(* IEC 61131-3 sources: SmartHomeNew/snapshots/2026-05-04 (part 2) *)

(* ---- FB_System_Timebase.st ---- *)
// ==============================================================================
// System timebase helper
//
// Internal helper for PRG_System.
// Owns PLC runtime clock projection into GVL_STATUS:
// - monotonic system milliseconds
// - time-of-day milliseconds
// - day of week / day of year rollover
// - TOD representation
// ==============================================================================
FUNCTION_BLOCK FB_System_Timebase
VAR
    L_Time_Diff : UDINT;
END_VAR

GVL_STATUS.G_System_Time_MS := TIME_TO_UDINT(TIME());

L_Time_Diff := SEL(
    GVL_STATUS.G_System_Time_MS >= GVL_STATUS.G_Last_System_Time_MS,
    GVL_STATUS.G_System_Time_MS - GVL_STATUS.G_Last_System_Time_MS,
    (4294967295 - GVL_STATUS.G_Last_System_Time_MS) + GVL_STATUS.G_System_Time_MS + 1
);

GVL_STATUS.G_Time_Of_Day_MS := (GVL_STATUS.G_Time_Of_Day_MS + L_Time_Diff) MOD 86400000;

IF GVL_STATUS.G_Time_Of_Day_MS < L_Time_Diff THEN
    GVL_STATUS.G_Current_Day := (GVL_STATUS.G_Current_Day MOD 7) + 1;
    GVL_STATUS.G_Day_Of_Year := (GVL_STATUS.G_Day_Of_Year MOD 365) + 1;
END_IF;

GVL_STATUS.G_Last_System_Time_MS := GVL_STATUS.G_System_Time_MS;
GVL_STATUS.G_Current_TOD := UDINT_TO_TOD(GVL_STATUS.G_Time_Of_Day_MS);

// >>> BULK_SYNC_ANCHOR: FB_System_Timebase <<<

(* ---- FB_Test_Result_Handler.st ---- *)
FUNCTION_BLOCK FB_Test_Result_Handler
VAR_INPUT
    VI_Test_Passed : BOOL;
END_VAR
VAR
    L_Latched_Failure : BOOL;
END_VAR

// latch failure
IF NOT VI_Test_Passed THEN
    L_Latched_Failure := TRUE;
END_IF;

// enforce safe stop if failure latched
IF L_Latched_Failure THEN
    GVL_COMMAND.G_Gas_Valve_Close := TRUE;
    GVL_COMMAND.G_Close_Valve_35 := TRUE;
    GVL_COMMAND.G_Close_Valve_36 := TRUE;
END_IF;
END_FUNCTION_BLOCK

(* ---- FB_Trend_Adapter.st ---- *)
FUNCTION_BLOCK FB_Trend_Adapter
VAR_INPUT
    VI_Data : ST_Trend_Data;
END_VAR

VAR_OUTPUT
    VO_Average : REAL;
    VO_Min : REAL;
    VO_Max : REAL;
    VO_Trend_Up : BOOL;
    VO_Trend_Down : BOOL;
END_VAR

VAR
    fbAnalyzer : FB_Trend_Analyzer;
    L_Data_Copy : ARRAY[1..GVL_CONSTANTS.C_MAX_TREND_DATA_POINTS] OF REAL;
    L_Count : INT;
    L_i : INT;
END_VAR

// Normalize count to analyzer bounds
L_Count := UDINT_TO_INT(VI_Data.record_count);
IF L_Count < 0 THEN
    L_Count := 0;
END_IF;
IF L_Count > GVL_CONSTANTS.C_MAX_TREND_DATA_POINTS THEN
    L_Count := GVL_CONSTANTS.C_MAX_TREND_DATA_POINTS;
END_IF;

// Copy source values into analyzer-compatible buffer
FOR L_i := 1 TO GVL_CONSTANTS.C_MAX_TREND_DATA_POINTS DO
    L_Data_Copy[L_i] := 0.0;
END_FOR;

IF L_Count > 0 THEN
    FOR L_i := 1 TO L_Count DO
        L_Data_Copy[L_i] := VI_Data.values[L_i];
    END_FOR;
END_IF;

fbAnalyzer(
    VI_Count := L_Count,
    VI_Data := L_Data_Copy,
    VO_Average => VO_Average,
    VO_Max => VO_Max,
    VO_Min => VO_Min,
    VO_Trend_Up => VO_Trend_Up,
    VO_Trend_Down => VO_Trend_Down
);
END_FUNCTION_BLOCK

(* ---- FB_Trend_Analyzer.st ---- *)
FUNCTION_BLOCK FB_Trend_Analyzer
VAR_INPUT
    VI_Count      : INT;
END_VAR
VAR_IN_OUT
    VI_Data       : ARRAY[1..GVL_CONSTANTS.C_MAX_TREND_DATA_POINTS] OF REAL;
END_VAR
VAR_OUTPUT
    VO_Average    : REAL;
    VO_Max        : REAL;
    VO_Min        : REAL;
    VO_Trend_Up   : BOOL;
    VO_Trend_Down : BOOL;
END_VAR
VAR
    L_i   : INT;
    L_Sum : REAL;
END_VAR

IF VI_Count > 0 AND VI_Count <= GVL_CONSTANTS.C_MAX_TREND_DATA_POINTS THEN
    VO_Max := VI_Data[1];
    VO_Min := VI_Data[1];
    L_Sum := 0.0;

    FOR L_i := 1 TO VI_Count DO
        IF VI_Data[L_i] > VO_Max THEN VO_Max := VI_Data[L_i]; END_IF;
        IF VI_Data[L_i] < VO_Min THEN VO_Min := VI_Data[L_i]; END_IF;
        L_Sum := L_Sum + VI_Data[L_i];
    END_FOR;

    VO_Average := L_Sum / INT_TO_REAL(VI_Count);

    IF VI_Count >= 2 THEN
        VO_Trend_Up := (VI_Data[VI_Count] > VI_Data[1]);
        VO_Trend_Down := (VI_Data[VI_Count] < VI_Data[1]);
    END_IF;
END_IF;
END_FUNCTION_BLOCK

(* ---- FB_Ventilation_System_Manager.st ---- *)
FUNCTION_BLOCK FB_Ventilation_System_Manager
VAR_INPUT
    VI_System_Time_MS : UDINT; // Системное время (мс)
    VI_IsActivePLC : BOOL; // Флаг: Данный ПЛК является ведущим
    VI_Outdoor_Temp : REAL; // Уличная температура воздуха (°C)
    VI_Current_Scenario : E_SCENARIO_TYPE; // Текущий глобальный сценарий
    VI_System_Mode : E_System_Operating_Mode; // Агрегированный режим работы системы
    VI_Config : ST_Ventilation_Global_Config; // Конфигурация системы вентиляции
    VI_Fire_Alarm : BOOL; // Сигнал пожарной тревоги
    VI_Gas_Alarm : BOOL; // Сигнал газовой тревоги
    VI_PV3_Boost_Req : BOOL; // Запрос форсирования ПВ-3 от газоанализатора (ТЗ 5.1)
    VI_Supply_100_Req : BOOL; // Запрос 100% притока (ТЗ 6.4)
    VI_Exhaust_100_Req : BOOL; // Запрос 100% вытяжки (ТЗ 6.4)
    VI_Supply_80_Req : BOOL; // Запрос 80% притока (ТЗ 5.4)
    VI_Vent_Stop : BOOL; // Запрос на остановку вентиляции (ТЗ 5.3)
    VI_IO_Modules_Online : ARRAY[1..GVL_CONSTANTS.C_MAX_MODULES] OF BOOL; // Статусы модулей ввода-вывода (только чтение)
END_VAR
VAR_IN_OUT
    VI_Supply_Temps : ARRAY[1..GVL_CONSTANTS.C_MAX_SUPPLY_TEMPS] OF REAL; // Температура приточного воздуха после калорифера
    VI_Room_Temps : ARRAY[1..16] OF REAL; // Температура в помещениях (°C)
    VI_Room_Humidities : ARRAY[1..16] OF REAL; // Влажность в помещениях (%)
    VI_Room_CO2 : ARRAY[1..16] OF REAL; // Уровень CO2 в помещениях (ppm)
    VI_Wet_Zone_Active : ARRAY[1..GVL_CONSTANTS.C_MAX_WET_ZONES] OF BOOL; // Сигналы включения света в санузлах (ТЗ 4.0)
    VI_Rule_Actions : ARRAY[1..GVL_CONSTANTS.C_MAX_RULES] OF ST_Rule_Action; // Действия от Rule Engine
END_VAR
VAR_OUTPUT
    VO_Supply_Fans : ARRAY[1..GVL_CONSTANTS.C_MAX_SUPPLY_FANS] OF BYTE; // Выход: Управление приточными вентиляторами (0-100%)
    VO_Exhaust_Fans : ARRAY[1..GVL_CONSTANTS.C_MAX_EXHAUST_FANS] OF BYTE; // Выход: Управление вытяжными вентиляторами (0-100%)
    VO_Heater_Power : ARRAY[1..GVL_CONSTANTS.C_MAX_BOILERS] OF REAL; // Выход: Мощность калориферов (0-100%)
    VO_Status_Msg : STRING(200); // Строковое сообщение о статусе
    VO_Ventilation_IO_Fault : BOOL; // Выход: диагностика потери связи с модулями ввода-вывода
    VO_Ventilation_Subsystem_Degraded : BOOL; // Выход: признак degraded-состояния подсистемы вентиляции
END_VAR
VAR
    L_Policy_Normal : BOOL;
    L_Policy_Safe_Stop : BOOL;
    L_Policy_Degraded : BOOL;
    L_Policy_Freeze_Protection : BOOL;
    L_i : INT;
    L_j : INT;
    L_Max_CO2 : REAL;
    L_Max_Hum : REAL;
    L_Base_Speed : BYTE;
    L_Target_Temp : REAL;
    L_PID_Heaters : ARRAY[1..GVL_CONSTANTS.C_MAX_BOILERS] OF FB_PID_Controller;
    L_Wet_Zone_Timers : ARRAY[1..GVL_CONSTANTS.C_MAX_WET_ZONES] OF FB_System_Timer_TOF; // Таймеры выбега для вытяжек санузлов
END_VAR

// ========================================
// Ventilation policy layer
// ========================================
VO_Ventilation_IO_Fault := FALSE;
VO_Ventilation_Subsystem_Degraded := FALSE;
L_Policy_Normal := (VI_System_Mode = E_System_Operating_Mode.MODE_NORMAL);
L_Policy_Safe_Stop := (VI_System_Mode = E_System_Operating_Mode.MODE_SAFE_STOP);
L_Policy_Degraded := (VI_System_Mode = E_System_Operating_Mode.MODE_DEGRADED);
L_Policy_Freeze_Protection := (VI_System_Mode = E_System_Operating_Mode.MODE_FREEZE_PROTECTION);

IF NOT VI_IsActivePLC THEN
    FOR L_i := 1 TO GVL_CONSTANTS.C_MAX_SUPPLY_FANS DO
        VO_Supply_Fans[L_i] := 0;
        IF L_i <= GVL_CONSTANTS.C_MAX_SUPPLY_TEMPS THEN
            VO_Heater_Power[L_i] := 0.0;
        END_IF;
    END_FOR;
    FOR L_i := 1 TO GVL_CONSTANTS.C_MAX_EXHAUST_FANS DO
        VO_Exhaust_Fans[L_i] := 0;
    END_FOR;
    VO_Status_Msg := 'ВЕНТИЛЯЦИЯ: РЕЗЕРВНЫЙ ПЛК';
    RETURN;
END_IF;

// Проверка связи с модулями ввода-вывода
FOR L_i := 1 TO GVL_CONSTANTS.C_MAX_MODULES DO
    IF NOT VI_IO_Modules_Online[L_i] THEN
        VO_Ventilation_IO_Fault := TRUE;
        // Переход в безопасное состояние при потере связи (отключение вентиляции)
        FOR L_j := 1 TO GVL_CONSTANTS.C_MAX_SUPPLY_FANS DO
            VO_Supply_Fans[L_j] := 0;
        END_FOR;
        FOR L_j := 1 TO GVL_CONSTANTS.C_MAX_EXHAUST_FANS DO
            VO_Exhaust_Fans[L_j] := 0;
        END_FOR;
        FOR L_j := 1 TO GVL_CONSTANTS.C_MAX_BOILERS DO
            VO_Heater_Power[L_j] := 0.0;
        END_FOR;
        VO_Status_Msg := 'ОШИБКА: Потеря связи с модулями ввода-вывода';
        RETURN;
    END_IF;
END_FOR;

// =========================
// SYSTEM MODE OVERRIDE
// =========================
// VENT_POLICY_ROUTING_PHASE3_V2
IF L_Policy_Safe_Stop THEN
    FOR L_i := 1 TO GVL_CONSTANTS.C_MAX_SUPPLY_FANS DO
        VO_Supply_Fans[L_i] := 0;
    END_FOR;
    FOR L_i := 1 TO GVL_CONSTANTS.C_MAX_EXHAUST_FANS DO
        VO_Exhaust_Fans[L_i] := 0;
    END_FOR;
    FOR L_i := 1 TO GVL_CONSTANTS.C_MAX_BOILERS DO
        VO_Heater_Power[L_i] := 0.0;
    END_FOR;
    VO_Status_Msg := 'ВЕНТИЛЯЦИЯ: ОСТАНОВЛЕНА POLICY SAFE_STOP';
    RETURN;
END_IF;

IF L_Policy_Degraded THEN
    FOR L_i := 1 TO GVL_CONSTANTS.C_MAX_SUPPLY_FANS DO
        VO_Supply_Fans[L_i] := 0;
    END_FOR;
    FOR L_i := 1 TO GVL_CONSTANTS.C_MAX_BOILERS DO
        VO_Heater_Power[L_i] := 0.0;
    END_FOR;
    VO_Ventilation_Subsystem_Degraded := TRUE;
    VO_Status_Msg := 'ВЕНТИЛЯЦИЯ: DEGRADED POLICY';
END_IF;

IF L_Policy_Freeze_Protection THEN
    FOR L_i := 1 TO GVL_CONSTANTS.C_MAX_SUPPLY_FANS DO
        VO_Supply_Fans[L_i] := 0;
    END_FOR;
    FOR L_i := 1 TO GVL_CONSTANTS.C_MAX_EXHAUST_FANS DO
        VO_Exhaust_Fans[L_i] := 0;
    END_FOR;
    FOR L_i := 1 TO GVL_CONSTANTS.C_MAX_BOILERS DO
        VO_Heater_Power[L_i] := 0.0;
    END_FOR;
    VO_Status_Msg := 'ВЕНТИЛЯЦИЯ: FREEZE_PROTECTION POLICY (stop)';
    RETURN;
END_IF;

// MODE_FREEZE_PROTECTION пока оставляем на текущей штатной логике

// 1. Определение базовой скорости и целевой температуры по сценарию (ТЗ 7.1)
CASE VI_Current_Scenario OF
    E_SCENARIO_TYPE.SCENARIO_AWAY:
        L_Base_Speed := VI_Config.Scenario_Modes[3].Base_Fan_Speed;
        L_Target_Temp := VI_Config.Scenario_Modes[3].Target_Temp;
    E_SCENARIO_TYPE.SCENARIO_SLEEP:
        L_Base_Speed := VI_Config.Scenario_Modes[2].Base_Fan_Speed;
        L_Target_Temp := VI_Config.Scenario_Modes[2].Target_Temp;
    ELSE // PRESENCE, MORNING, EVENING
        L_Base_Speed := VI_Config.Scenario_Modes[1].Base_Fan_Speed;
        L_Target_Temp := VI_Config.Scenario_Modes[1].Target_Temp;
END_CASE;

// 2. Логика управления приточными установками (П-1, П-2, П-3)
FOR L_i := 1 TO GVL_CONSTANTS.C_MAX_SUPPLY_FANS DO
    // ПИД-регулирование мощности электрического калорифера
    IF L_i <= GVL_CONSTANTS.C_MAX_SUPPLY_TEMPS THEN
        L_PID_Heaters[L_i](
            VI_SetPoint := L_Target_Temp,
            VI_ProcessValue := VI_Supply_Temps[L_i], // Используем датчик температуры после калорифера
            VI_Kp := 4.0, VI_Tn := 120.0, VI_Tv := 0.0,
            VI_Y_Min := 0.0, VI_Y_Max := 100.0, VI_Cycle_Time_S := 1.0,
            VO_Output => VO_Heater_Power[L_i]
        );
    END_IF;

    // Определение скорости приточного вентилятора
    VO_Supply_Fans[L_i] := L_Base_Speed;

    // Обработка действий от Rule Engine
    FOR L_j := 1 TO GVL_CONSTANTS.C_MAX_RULES DO
        IF VI_Rule_Actions[L_j].Active AND VI_Rule_Actions[L_j].Target_ID = L_i THEN
            IF VI_Rule_Actions[L_j].Action_Type = E_Rule_Action_Type.ACTION_SET_VENTILATION THEN
                VO_Supply_Fans[L_i] := REAL_TO_BYTE(VI_Rule_Actions[L_j].Value);
            END_IF;
        END_IF;
    END_FOR;

    // Requests are operational requests and must not be reported as subsystem degradation.
END_FOR;

// 3. Логика управления вытяжными установками (В-1 .. В-5)
FOR L_i := 1 TO GVL_CONSTANTS.C_MAX_EXHAUST_FANS DO
    VO_Exhaust_Fans[L_i] := L_Base_Speed;

    // ТЗ 4.0: Логика вытяжки в санузлах
    FOR L_j := 1 TO GVL_CONSTANTS.C_MAX_WET_ZONES DO
        IF VI_Config.wet_zone_to_exhaust_map[L_j] = L_i THEN
            // Включение по свету, выключение с задержкой 5 минут (используем TOF)
            L_Wet_Zone_Timers[L_j](IN := VI_Wet_Zone_Active[L_j], PT := T#5m, VI_System_Time_MS := VI_System_Time_MS);
            IF VI_Wet_Zone_Active[L_j] THEN
                VO_Exhaust_Fans[L_i] := 80; // Повышенная скорость при присутствии
            ELSIF L_Wet_Zone_Timers[L_j].Q THEN
                VO_Exhaust_Fans[L_i] := 50; // Скорость выбега (пока таймер TOF активен)
            END_IF;
        END_IF;
    END_FOR;

    // Requests are operational requests and must not be reported as subsystem degradation.
END_FOR;

// ========================================
// VENT_FINAL_CLAMP
// ========================================
IF L_Policy_Degraded THEN
    FOR L_i := 1 TO GVL_CONSTANTS.C_MAX_EXHAUST_FANS DO
        VO_Exhaust_Fans[L_i] := MIN(VO_Exhaust_Fans[L_i], VI_Config.Degraded_Exhaust_Limit);
    END_FOR;
END_IF;

// 4. Формирование статусного сообщения
IF L_Policy_Safe_Stop THEN
    VO_Status_Msg := 'ВЕНТИЛЯЦИЯ: ОСТАНОВЛЕНА POLICY SAFE_STOP';
ELSIF L_Policy_Freeze_Protection THEN
    VO_Status_Msg := 'ВЕНТИЛЯЦИЯ: FREEZE_PROTECTION POLICY (stop)';
ELSIF L_Policy_Degraded THEN
    VO_Status_Msg := 'ВЕНТИЛЯЦИЯ: DEGRADED POLICY';
ELSE
    VO_Status_Msg := 'Вентиляция работает в штатном режиме';
END_IF;
// >>> BULK_SYNC_ANCHOR: FB_Ventilation_System_Manager <<<

(* ---- FB_Water_Leakage_Manager.st ---- *)
FUNCTION_BLOCK FB_Water_Leakage_Manager
VAR_INPUT
    VI_System_Time_MS : UDINT;
    VI_IsActivePLC    : BOOL;
    VI_Config         : ST_Flood_Global_Config;
END_VAR

VAR_IN_OUT
    VI_Sensors : ARRAY[1..GVL_CONSTANTS.C_MAX_FLOOD_SENSORS] OF BOOL;
END_VAR

VAR_OUTPUT
    VO_Status_Msg     : STRING(200);
    VO_Leak_Detected      : BOOL;
    VO_Leak_Warning_Level : BOOL;
END_VAR

VAR
    L_i             : INT;
    L_Sensor_Timers : ARRAY[1..GVL_CONSTANTS.C_MAX_FLOOD_SENSORS] OF FB_System_Timer;
    L_Any_Leak      : BOOL;
    L_Any_Warning   : BOOL;
END_VAR

IF NOT VI_IsActivePLC THEN RETURN; END_IF;

L_Any_Leak := FALSE;
L_Any_Warning := FALSE;

FOR L_i := 1 TO GVL_CONSTANTS.C_MAX_FLOOD_SENSORS DO
    L_Sensor_Timers[L_i](
        IN := VI_Sensors[L_i],
        PT := TO_TIME(VI_Config.min_duration_ms + VI_Config.warning_duration_ms),
        VI_System_Time_MS := VI_System_Time_MS
    );

    IF L_Sensor_Timers[L_i].ET >= TO_TIME(VI_Config.min_duration_ms) THEN
        L_Any_Warning := TRUE;

        IF L_Sensor_Timers[L_i].Q THEN
            L_Any_Leak := TRUE;
        END_IF;
    END_IF;
END_FOR;

// Manual latch instead of RS
IF GVL_INTENT_USER.I_Reset_Errors THEN
    VO_Leak_Detected := FALSE;
ELSIF L_Any_Leak THEN
    VO_Leak_Detected := TRUE;
END_IF;

VO_Leak_Warning_Level := L_Any_Warning;

IF VO_Leak_Detected THEN
    VO_Status_Msg := 'АВАРИЯ: ПРОТЕЧКА ВОДЫ.';
ELSIF L_Any_Warning THEN
    VO_Status_Msg := 'ПРЕДУПРЕЖДЕНИЕ: ОБНАРУЖЕНА ВОДА.';
ELSE
    VO_Status_Msg := 'Система контроля протечек в норме';
END_IF;
// >>> BULK_SYNC_ANCHOR: FB_Water_Leakage_Manager <<<

(* ---- MAIN.st ---- *)
PROGRAM MAIN

PRG_Time_Service();
PRG_System_Init();
PRG_PLC_Arbitration();
PRG_Config_Manager();
PRG_Config_Validation();
PRG_Config_Versioning();
PRG_IO_Read();
PRG_Input_Processing();
PRG_User_Adapt_Control();
PRG_Behavior_Adapt_Profile();
PRG_Safety();
PRG_Safety_Operator();
PRG_Safety_Shutdown();
PRG_Safety_Recovery();
PRG_System_Intent();
PRG_System_Health();
PRG_System_Alarm_Gateway();
PRG_System_Scenario_Rules();
PRG_System_Access_Maintenance();
PRG_System_BlackBox();
PRG_System_History();
PRG_System_Diagnostics();
PRG_System_Diagnostics_Ext();
PRG_System_Evacuation();
PRG_System_Trend();
PRG_System_Runtime_Base();
PRG_Presence_Manager();
PRG_System_Simulation();
PRG_Heating_Policy_Manager();
PRG_Heating_Policy_Observer();
PRG_Mode_Manager();
PRG_System_Coordinator();
PRG_Policy();
PRG_Scenario_Engine();
PRG_Command_Arbitration();
PRG_Command_Verifier();
PRG_Security();
PRG_Heating();
PRG_Ventilation();
PRG_Lighting();
PRG_Water();
PRG_Access();
PRG_Explainability();
PRG_HMI_Dashboard();
PRG_Debug_View();
PRG_IO_Write();
END_PROGRAM

(* ---- PRG_Access.st ---- *)
PROGRAM PRG_Access
VAR
    fbProjection : FB_Access_Output_Projection;
END_VAR

fbProjection(
    VI_Lock_1_Open := GVL_COMMAND_SHADOW.G_Lock_1_Open,
    VI_Lock_1_Close := GVL_COMMAND_SHADOW.G_Lock_1_Close,
    VI_Lock_2_Open := GVL_COMMAND_SHADOW.G_Lock_2_Open,
    VI_Lock_2_Close := GVL_COMMAND_SHADOW.G_Lock_2_Close,
    VI_Gate_Open := GVL_COMMAND_SHADOW.G_Gate_Open,
    VI_Wicket_Open := GVL_COMMAND_SHADOW.G_Wicket_Open
);

// >>> BULK_SYNC_ANCHOR: PRG_Access <<<
END_PROGRAM

(* ---- PRG_Behavior_Adapt_Profile.st ---- *)
PROGRAM PRG_Behavior_Adapt_Profile

// Centralized tuning profile controller.
// This block enforces consistent adaptive behavior settings.

CASE GVL_BEHAVIOR_ADAPT.G_Adapt_Profile OF

    ADAPT_PROFILE_STABLE:
        GVL_BEHAVIOR_ADAPT.G_Adapt_Learning_Rate := 0.03;
        GVL_BEHAVIOR_ADAPT.G_Confidence_Learning_Rate := 0.03;
        GVL_BEHAVIOR_ADAPT.G_Decay_Factor := 0.998;
        GVL_BEHAVIOR_ADAPT.G_Adapt_Update_Threshold := 7;

    ADAPT_PROFILE_BALANCED:
        GVL_BEHAVIOR_ADAPT.G_Adapt_Learning_Rate := 0.05;
        GVL_BEHAVIOR_ADAPT.G_Confidence_Learning_Rate := 0.05;
        GVL_BEHAVIOR_ADAPT.G_Decay_Factor := 0.995;
        GVL_BEHAVIOR_ADAPT.G_Adapt_Update_Threshold := 5;

    ADAPT_PROFILE_AGGRESSIVE:
        GVL_BEHAVIOR_ADAPT.G_Adapt_Learning_Rate := 0.08;
        GVL_BEHAVIOR_ADAPT.G_Confidence_Learning_Rate := 0.08;
        GVL_BEHAVIOR_ADAPT.G_Decay_Factor := 0.990;
        GVL_BEHAVIOR_ADAPT.G_Adapt_Update_Threshold := 3;

ELSE
        // No fallback required
END_CASE;

// >>> BULK_SYNC_ANCHOR: PRG_Behavior_Adapt_Profile <<<
END_PROGRAM

(* ---- PRG_Command_Verifier.st ---- *)
PROGRAM PRG_Command_Verifier
VAR
    L_Mismatch_Count : INT := 0;
END_VAR

// Current-cycle mismatch count between legacy and shadow command layers
L_Mismatch_Count := 0;

IF GVL_COMMAND.G_Gas_Valve_Close <> GVL_COMMAND_SHADOW.G_Gas_Valve_Close THEN
    L_Mismatch_Count := L_Mismatch_Count + 1;
END_IF;

IF GVL_COMMAND.G_Boiler_Stop <> GVL_COMMAND_SHADOW.G_Boiler_Stop THEN
    L_Mismatch_Count := L_Mismatch_Count + 1;
END_IF;

IF GVL_COMMAND.G_Vent_Stop <> GVL_COMMAND_SHADOW.G_Vent_Stop THEN
    L_Mismatch_Count := L_Mismatch_Count + 1;
END_IF;

IF GVL_COMMAND.G_Supply_100_Req <> GVL_COMMAND_SHADOW.G_Supply_100_Req THEN
    L_Mismatch_Count := L_Mismatch_Count + 1;
END_IF;

IF GVL_COMMAND.G_Supply_80_Req <> GVL_COMMAND_SHADOW.G_Supply_80_Req THEN
    L_Mismatch_Count := L_Mismatch_Count + 1;
END_IF;

IF GVL_COMMAND.G_Vent_PV3_Boost <> GVL_COMMAND_SHADOW.G_Vent_PV3_Boost THEN
    L_Mismatch_Count := L_Mismatch_Count + 1;
END_IF;

IF GVL_COMMAND.G_Close_Valve_35 <> GVL_COMMAND_SHADOW.G_Close_Valve_35 THEN
    L_Mismatch_Count := L_Mismatch_Count + 1;
END_IF;

IF GVL_COMMAND.G_Close_Valve_36 <> GVL_COMMAND_SHADOW.G_Close_Valve_36 THEN
    L_Mismatch_Count := L_Mismatch_Count + 1;
END_IF;

IF GVL_COMMAND.G_Lock_1_Open <> GVL_COMMAND_SHADOW.G_Lock_1_Open THEN
    L_Mismatch_Count := L_Mismatch_Count + 1;
END_IF;

IF GVL_COMMAND.G_Lock_1_Close <> GVL_COMMAND_SHADOW.G_Lock_1_Close THEN
    L_Mismatch_Count := L_Mismatch_Count + 1;
END_IF;

IF GVL_COMMAND.G_Lock_2_Open <> GVL_COMMAND_SHADOW.G_Lock_2_Open THEN
    L_Mismatch_Count := L_Mismatch_Count + 1;
END_IF;

IF GVL_COMMAND.G_Lock_2_Close <> GVL_COMMAND_SHADOW.G_Lock_2_Close THEN
    L_Mismatch_Count := L_Mismatch_Count + 1;
END_IF;

// Gate and wicket comparison
IF GVL_COMMAND.G_Gate_Open <> GVL_COMMAND_SHADOW.G_Gate_Open THEN
    L_Mismatch_Count := L_Mismatch_Count + 1;
END_IF;

IF GVL_COMMAND.G_Wicket_Open <> GVL_COMMAND_SHADOW.G_Wicket_Open THEN
    L_Mismatch_Count := L_Mismatch_Count + 1;
END_IF;

GVL_COMMAND_VERIFY.Command_Mismatch_Count := L_Mismatch_Count;
GVL_COMMAND_VERIFY.Command_Match_OK := (L_Mismatch_Count = 0);
GVL_COMMAND_VERIFY.Command_Mismatch_Active := (L_Mismatch_Count > 0);

(* ---- PRG_Config_Simulation.st ---- *)
PROGRAM PRG_Config_Simulation
VAR
    L_Error : BOOL;
END_VAR

L_Error := FALSE;
GVL_CONFIG_SIMULATION.G_Simulation_Result_OK := TRUE;
GVL_CONFIG_SIMULATION.G_Simulation_Error_Text := '';

IF GVL_CONFIG_SIMULATION.G_Simulation_Request AND GVL_CONFIG_SIMULATION.G_Simulation_Confirm THEN

    // Simulate INPUT constraints
    IF (GVL_CONFIG_CONTROL.STG_Reputation_Learning_Rate < 0.0) OR (GVL_CONFIG_CONTROL.STG_Reputation_Learning_Rate > 1.0) THEN
        GVL_CONFIG_SIMULATION.G_Simulation_Result_OK := FALSE;
        GVL_CONFIG_SIMULATION.G_Simulation_Error_Text := 'Invalid learning rate';
        L_Error := TRUE;
    END_IF;

    // Simulate SCENARIO logic
    IF GVL_CONFIG_CONTROL.STG_Night_Start_Hour = GVL_CONFIG_CONTROL.STG_Night_End_Hour THEN
        GVL_CONFIG_SIMULATION.G_Simulation_Result_OK := FALSE;
        GVL_CONFIG_SIMULATION.G_Simulation_Error_Text := 'Night window invalid';
        L_Error := TRUE;
    END_IF;

    // Simulate SAFETY
    IF GVL_CONFIG_CONTROL.STG_Stabilization_Delay_MS < 1000 THEN
        GVL_CONFIG_SIMULATION.G_Simulation_Result_OK := FALSE;
        GVL_CONFIG_SIMULATION.G_Simulation_Error_Text := 'Recovery delay too small';
        L_Error := TRUE;
    END_IF;

    // Simulate FAIL-SAFE policy
    IF NOT (
        GVL_CONFIG_CONTROL.STG_PLC_Inactive_Close_Gas OR
        GVL_CONFIG_CONTROL.STG_PLC_Inactive_Stop_Boiler OR
        GVL_CONFIG_CONTROL.STG_PLC_Inactive_Block_Heating OR
        GVL_CONFIG_CONTROL.STG_PLC_Inactive_Stop_Vent OR
        GVL_CONFIG_CONTROL.STG_PLC_Inactive_Block_Water
    ) THEN
        GVL_CONFIG_SIMULATION.G_Simulation_Result_OK := FALSE;
        GVL_CONFIG_SIMULATION.G_Simulation_Error_Text := 'Fail-safe disabled';
        L_Error := TRUE;
    END_IF;

    GVL_CONFIG_SIMULATION.G_Simulation_Last_Run_MS := GVL_TIME_SERVICE.G_Now_MS;

END_IF;

// >>> BULK_SYNC_ANCHOR: PRG_Config_Simulation <<<

(* ---- PRG_Config_Validation.st ---- *)
PROGRAM PRG_Config_Validation
VAR
    L_i : INT;
    L_Zone : INT;
    L_Sensor : INT;
    L_Manifold : INT;
    L_Config_Error : BOOL;
END_VAR

L_Config_Error := FALSE;

FOR L_i := 1 TO GVL_CONSTANTS.C_MAX_HEATING_CIRCUITS DO
    L_Zone := BYTE_TO_INT(GVL_CONFIG.G_HMI_FloorHeating_Configs[L_i].zone);
    L_Sensor := BYTE_TO_INT(GVL_CONFIG.G_HMI_FloorHeating_Configs[L_i].sensor_id);
    L_Manifold := BYTE_TO_INT(GVL_CONFIG.G_HMI_FloorHeating_Configs[L_i].manifold_id);

    IF (L_Zone < 1) OR (L_Zone > GVL_CONSTANTS.C_MAX_ZONES) THEN
        L_Config_Error := TRUE;
    END_IF;

    IF (L_Sensor < 1) OR (L_Sensor > GVL_CONSTANTS.C_MAX_ZONES) THEN
        L_Config_Error := TRUE;
    END_IF;

    IF (L_Manifold < 1) OR (L_Manifold > GVL_CONSTANTS.C_MAX_MANIFOLDS) THEN
        L_Config_Error := TRUE;
    END_IF;

    IF GVL_CONFIG.G_HMI_FloorHeating_Configs[L_i].min_temp > GVL_CONFIG.G_HMI_FloorHeating_Configs[L_i].max_temp THEN
        L_Config_Error := TRUE;
    END_IF;

    IF (GVL_CONFIG.G_HMI_FloorHeating_Configs[L_i].design_temp < GVL_CONFIG.G_HMI_FloorHeating_Configs[L_i].min_temp) OR
       (GVL_CONFIG.G_HMI_FloorHeating_Configs[L_i].design_temp > GVL_CONFIG.G_HMI_FloorHeating_Configs[L_i].max_temp) THEN
        L_Config_Error := TRUE;
    END_IF;
END_FOR;

IF GVL_CONFIG.G_Max_Active_Manifolds < 1 THEN
    L_Config_Error := TRUE;
ELSIF GVL_CONFIG.G_Max_Active_Manifolds > GVL_CONSTANTS.C_MAX_MANIFOLDS THEN
    L_Config_Error := TRUE;
END_IF;

IF GVL_CONFIG.G_Max_Thermal_Budget <= 0.0 THEN
    L_Config_Error := TRUE;
END_IF;

IF L_Config_Error THEN
    GVL_STATUS.G_Diagnostics.Sensor_Fault := TRUE;
    GVL_STATUS.G_Diagnostics.Subsystem_Degraded := TRUE;
    GVL_STATUS.G_System_Mode_Text := 'CONFIG ERROR';
    GVL_COMMAND_SHADOW.G_Heating_Block := TRUE;
    GVL_COMMAND_SHADOW.G_Boiler_Stop := TRUE;
END_IF;

END_PROGRAM
// >>> BULK_SYNC_ANCHOR: PRG_Config_Validation <<<

(* ---- PRG_Heating.st ---- *)
PROGRAM PRG_Heating
VAR
    fbLocalContext : FB_Heating_Local_Context;
    fbThermalAllocation : FB_Heating_Thermal_Allocation;
    fbHeatingOrchestration : FB_Heating_Orchestration;
    fbHeatingDiagnostics : FB_Heating_Diagnostics;
    fbHeatingMaintenanceGating : FB_Heating_Maintenance_Gating;
    fbHeatingFreezeHardware : FB_Heating_Freeze_Hardware;
    fbHeatingRootCauseDiagnostics : FB_Heating_RootCause_Diagnostics;
    fbOutputProjection : FB_Heating_Output_Projection;
    L_i : INT;
    L_Zone_Index : INT;
    L_Manifold_Index : INT;
    L_Sensor_Index : INT;
    L_Config_Mapping_Error : BOOL;
    L_Outdoor_Temp : REAL;
    L_Room_Temps : ARRAY[1..GVL_CONSTANTS.C_MAX_ZONES] OF REAL;
    L_Floor_Temps : ARRAY[1..GVL_CONSTANTS.C_MAX_HEATING_CIRCUITS] OF REAL;
    L_Manifold_Pressures : ARRAY[1..GVL_CONSTANTS.C_MAX_MANIFOLDS] OF REAL;
    L_Zone_Configs : ARRAY[1..GVL_CONSTANTS.C_MAX_HEATING_CIRCUITS] OF ST_FloorHeating_Circuit_Config;
    L_Circuit_To_Zone : ARRAY[1..GVL_CONSTANTS.C_MAX_HEATING_CIRCUITS] OF INT;
    L_Zone_Valves : ARRAY[1..GVL_CONSTANTS.C_MAX_HEATING_CIRCUITS] OF BOOL;
    L_Manifold_Pumps : ARRAY[1..GVL_CONSTANTS.C_MAX_MANIFOLDS] OF BOOL;
    L_Manifold_Valves : ARRAY[1..GVL_CONSTANTS.C_MAX_MANIFOLDS] OF REAL;
    L_Boiler_OT_Enable : ARRAY[1..GVL_CONSTANTS.C_MAX_BOILERS] OF BOOL;
    L_Boiler_OT_Setpoint : ARRAY[1..GVL_CONSTANTS.C_MAX_BOILERS] OF REAL;
    L_Backup_Circulation_Pump : BOOL;
    L_Electric_Heater_Enable : BOOL;
    L_Freeze_Risk_Status : BOOL;
    L_Manifold_Status : ARRAY[1..GVL_CONSTANTS.C_MAX_MANIFOLDS] OF ST_Manifold_Status;
    L_Boiler_Status : ARRAY[1..GVL_CONSTANTS.C_MAX_BOILERS] OF ST_Boiler_Status;
    L_DHW_Heating_Pump : BOOL;
    L_DHW_Circ_Pump : BOOL;
    L_DHW_Status : ST_DHW_Status;
END_VAR

IF (GVL_STATE.G_Outdoor_Temp > -50.0) AND (GVL_STATE.G_Outdoor_Temp < 60.0) THEN
    L_Outdoor_Temp := LIMIT(-50.0, GVL_STATE.G_Outdoor_Temp, 60.0);
ELSE
    L_Outdoor_Temp := 0.0;
END_IF;

FOR L_i := 1 TO GVL_CONSTANTS.C_MAX_ZONES DO
    IF (GVL_STATE.G_Room_Temps[L_i] > -50.0) AND (GVL_STATE.G_Room_Temps[L_i] < 100.0) THEN
        L_Room_Temps[L_i] := GVL_STATE.G_Room_Temps[L_i];
    ELSE
        L_Room_Temps[L_i] := 20.0;
    END_IF;
END_FOR;

FOR L_i := 1 TO GVL_CONSTANTS.C_MAX_HEATING_CIRCUITS DO
    IF (GVL_STATE.G_Floor_Temps[L_i] > -50.0) AND (GVL_STATE.G_Floor_Temps[L_i] < 100.0) THEN
        L_Floor_Temps[L_i] := GVL_STATE.G_Floor_Temps[L_i];
    ELSE
        L_Floor_Temps[L_i] := 20.0;
    END_IF;
END_FOR;

FOR L_i := 1 TO GVL_CONSTANTS.C_MAX_MANIFOLDS DO
    IF (GVL_STATE.G_Manifold_Pressures[L_i] > 0.1) THEN
        L_Manifold_Pressures[L_i] := GVL_STATE.G_Manifold_Pressures[L_i];
    ELSE
        L_Manifold_Pressures[L_i] := 0.0;
    END_IF;
END_FOR;

// rest unchanged
// >>> BULK_SYNC_ANCHOR: PRG_Heating <<<

(* ---- PRG_IO_Read.st ---- *)
PROGRAM PRG_IO_Read
VAR
    L_i : INT;
    L_Debounce_Time : TIME := T#100MS;
    L_Manifold_Pressure_Raw : WORD;
    L_Manifold_Current_Raw : WORD;
    L_Filtered_Room_Temp : REAL;
    L_Filtered_Floor_Temp : REAL;

    fbDebounce_Switches : ARRAY[1..8] OF FB_System_Timer;
    fbDebounce_Motion : ARRAY[1..8] OF FB_System_Timer;
    fbDebounce_Security_Open : ARRAY[1..GVL_CONSTANTS.C_MAX_SECURITY_SENSORS] OF FB_System_Timer;
    fbDebounce_Security_Glass : ARRAY[1..GVL_CONSTANTS.C_MAX_SECURITY_SENSORS] OF FB_System_Timer;
    fbDebounce_Flood : ARRAY[1..GVL_CONSTANTS.C_MAX_FLOOD_SENSORS] OF FB_System_Timer;
    fbDebounce_Smoke : ARRAY[1..GVL_CONSTANTS.C_MAX_SMOKE_SENSORS] OF FB_System_Timer;
    fbDebounce_Group_2F : FB_System_Timer;

    fbIO_Watchdog_1 : FB_IO_Module_Watchdog;
    fbIO_Watchdog_2 : FB_IO_Module_Watchdog;
    fbDiagEventManager : FB_Diagnostics_Event_Manager;
    L_IO_Error_Active : BOOL;

    fbCalib_Outdoor_Temp : FB_Sensor_Calibration_Processor;
    fbCalib_Supply_Temps : ARRAY[1..GVL_CONSTANTS.C_MAX_SUPPLY_TEMPS] OF FB_Sensor_Calibration_Processor;
    fbCalib_Room_Temps : ARRAY[1..GVL_CONSTANTS.C_MAX_ZONES] OF FB_Sensor_Calibration_Processor;
    fbCalib_Floor_Temps : ARRAY[1..GVL_CONSTANTS.C_MAX_ZONES] OF FB_Sensor_Calibration_Processor;
    fbCalib_Room_Hum : ARRAY[1..GVL_CONSTANTS.C_MAX_ZONES] OF FB_Sensor_Calibration_Processor;
    fbCalib_Room_CO2 : ARRAY[1..GVL_CONSTANTS.C_MAX_ZONES] OF FB_Sensor_Calibration_Processor;
    fbCalib_Manifold_T_Supply : ARRAY[1..GVL_CONSTANTS.C_MAX_MANIFOLDS] OF FB_Sensor_Calibration_Processor;
    fbCalib_Manifold_T_Return : ARRAY[1..GVL_CONSTANTS.C_MAX_MANIFOLDS] OF FB_Sensor_Calibration_Processor;
    fbCalib_Methane : ARRAY[1..GVL_CONSTANTS.C_MAX_METHANE_SENSORS] OF FB_Sensor_Calibration_Processor;
    fbCalib_CO : ARRAY[1..GVL_CONSTANTS.C_MAX_CO_SENSORS] OF FB_Sensor_Calibration_Processor;

    fbAnalog_Manifold_Pressure : ARRAY[1..GVL_CONSTANTS.C_MAX_MANIFOLDS] OF FB_Sensor_Analog_Processing;
    fbAnalog_Manifold_Current : ARRAY[1..GVL_CONSTANTS.C_MAX_MANIFOLDS] OF FB_Sensor_Analog_Processing;
END_VAR

fbIO_Watchdog_1(VI_System_Time_MS := GVL_STATUS.G_System_Time_MS, VI_Module_ID := 1, VI_Heartbeat_Signal := GVL_IO.DI_Module_1_Heartbeat, VI_Timeout_MS := 2000);
fbIO_Watchdog_2(VI_System_Time_MS := GVL_STATUS.G_System_Time_MS, VI_Module_ID := 2, VI_Heartbeat_Signal := GVL_IO.DI_Module_2_Heartbeat, VI_Timeout_MS := 2000);

GVL_STATUS.G_IO_Modules_Online[1] := fbIO_Watchdog_1.VO_Module_Online;
GVL_STATUS.G_IO_Modules_Online[2] := fbIO_Watchdog_2.VO_Module_Online;

L_IO_Error_Active := fbIO_Watchdog_1.VO_Error_Active OR fbIO_Watchdog_2.VO_Error_Active;

fbDiagEventManager(
    VI_Code := 16#E001,
    VI_Severity := 4,
    VI_Active := NOT fbIO_Watchdog_1.VO_Module_Online,
    VI_Timestamp := GVL_STATUS.G_System_Time_MS,
    VI_Source := 1,
    VIO_Events := GVL_STATUS.G_Diagnostics_Events,
    VIO_Count := GVL_STATUS.G_Diagnostics_Count
);

fbDiagEventManager(
    VI_Code := 16#E002,
    VI_Severity := 4,
    VI_Active := NOT fbIO_Watchdog_2.VO_Module_Online,
    VI_Timestamp := GVL_STATUS.G_System_Time_MS,
    VI_Source := 2,
    VIO_Events := GVL_STATUS.G_Diagnostics_Events,
    VIO_Count := GVL_STATUS.G_Diagnostics_Count
);

IF L_IO_Error_Active THEN
    FOR L_i := 1 TO GVL_CONSTANTS.C_MAX_MANIFOLDS DO
        GVL_STATE.G_Manifold_Pumps[L_i] := FALSE;
    END_FOR;
END_IF;

FOR L_i := 1 TO 8 DO
    fbDebounce_Switches[L_i](IN := GVL_IO.DI_Lighting_Switches[L_i], PT := L_Debounce_Time, VI_System_Time_MS := GVL_STATUS.G_System_Time_MS);
    GVL_STATE.G_Physical_Switches[L_i] := fbDebounce_Switches[L_i].Q;

    fbDebounce_Motion[L_i](IN := GVL_IO.DI_Motion_Sensors[L_i], PT := L_Debounce_Time, VI_System_Time_MS := GVL_STATUS.G_System_Time_MS);
    GVL_STATE.G_Motion_Sensors[L_i] := fbDebounce_Motion[L_i].Q;
END_FOR;

FOR L_i := 1 TO GVL_CONSTANTS.C_MAX_SOCKETS DO
    GVL_STATE.G_Socket_Switches[L_i] := FALSE;
END_FOR;

FOR L_i := 1 TO GVL_CONSTANTS.C_MAX_SECURITY_SENSORS DO
    fbDebounce_Security_Open[L_i](IN := GVL_IO.DI_Security_Open[L_i], PT := L_Debounce_Time, VI_System_Time_MS := GVL_STATUS.G_System_Time_MS);
    fbDebounce_Security_Glass[L_i](IN := GVL_IO.DI_Security_Glass[L_i], PT := L_Debounce_Time, VI_System_Time_MS := GVL_STATUS.G_System_Time_MS);
END_FOR;

fbDebounce_Group_2F(IN := GVL_IO.DI_Security_2F_Group, PT := L_Debounce_Time, VI_System_Time_MS := GVL_STATUS.G_System_Time_MS);

FOR L_i := 1 TO GVL_CONSTANTS.C_MAX_DOOR_SENSORS DO
    IF GVL_CONFIG.G_Door_Map[L_i] > 0 AND GVL_CONFIG.G_Door_Map[L_i] <= GVL_CONSTANTS.C_MAX_SECURITY_SENSORS THEN
        GVL_STATE.G_Door_Sensors[L_i] := fbDebounce_Security_Open[GVL_CONFIG.G_Door_Map[L_i]].Q;
    END_IF;
END_FOR;

FOR L_i := 1 TO 8 DO
    IF GVL_CONFIG.G_Window_Map[L_i] > 0 THEN
        IF GVL_CONFIG.G_Window_Map[L_i] <= GVL_CONSTANTS.C_MAX_SECURITY_SENSORS THEN
            GVL_STATE.G_Window_Sensors[L_i] := fbDebounce_Security_Open[GVL_CONFIG.G_Window_Map[L_i]].Q;
        ELSE
            GVL_STATE.G_Window_Sensors[L_i] := fbDebounce_Security_Glass[GVL_CONFIG.G_Window_Map[L_i] - GVL_CONSTANTS.C_MAX_SECURITY_SENSORS].Q;
        END_IF;
    END_IF;
END_FOR;
GVL_STATE.G_Window_Sensors[16] := fbDebounce_Group_2F.Q;

FOR L_i := 1 TO GVL_CONSTANTS.C_MAX_FLOOD_SENSORS DO
    fbDebounce_Flood[L_i](IN := GVL_IO.DI_Flood_Sensors[L_i], PT := L_Debounce_Time, VI_System_Time_MS := GVL_STATUS.G_System_Time_MS);
    GVL_STATE.G_Water_Sensors[L_i] := fbDebounce_Flood[L_i].Q;
END_FOR;

FOR L_i := 1 TO GVL_CONSTANTS.C_MAX_SMOKE_SENSORS DO
    fbDebounce_Smoke[L_i](IN := GVL_IO.DI_Smoke_Sensors[L_i], PT := L_Debounce_Time, VI_System_Time_MS := GVL_STATUS.G_System_Time_MS);
    GVL_STATE.G_Smoke_Sensors[L_i] := fbDebounce_Smoke[L_i].Q;
END_FOR;

fbCalib_Outdoor_Temp(
    VI_Raw_Value := GVL_IO.AI_Temp_Outdoor.rValue,
    VI_Record := GVL_CONFIG.G_Calib_Outdoor_Temp
);
GVL_STATE.G_Outdoor_Temp := fbCalib_Outdoor_Temp.VO_Calibrated_Value;

FOR L_i := 1 TO GVL_CONSTANTS.C_MAX_SUPPLY_TEMPS DO
    IF GVL_IO.AI_Supply_Temps[L_i].wStatus = 0 THEN
        fbCalib_Supply_Temps[L_i](
            VI_Raw_Value := GVL_IO.AI_Supply_Temps[L_i].rValue,
            VI_Record := GVL_CONFIG.G_Calib_Supply_Temps[L_i]
        );
        GVL_STATE.G_Supply_Temps[L_i] := fbCalib_Supply_Temps[L_i].VO_Calibrated_Value;
    END_IF;
END_FOR;

FOR L_i := 1 TO 8 DO
    fbCalib_Room_Hum[L_i](
        VI_Raw_Value := GVL_IO.AI_Room_Hum[L_i],
        VI_Record := GVL_CONFIG.G_Calib_Humidity[L_i]
    );
    GVL_STATE.G_Room_Hum[L_i] := fbCalib_Room_Hum[L_i].VO_Calibrated_Value;

    fbCalib_Room_CO2[L_i](
        VI_Raw_Value := GVL_IO.AI_Room_CO2[L_i],
        VI_Record := GVL_CONFIG.G_Calib_CO2[L_i]
    );
    GVL_STATE.G_Room_CO2[L_i] := fbCalib_Room_CO2[L_i].VO_Calibrated_Value;
END_FOR;

// Room temperature filtering and range validation
FOR L_i := 1 TO GVL_CONSTANTS.C_MAX_ZONES DO
    fbCalib_Room_Temps[L_i](
        VI_Raw_Value := GVL_IO.AI_Room_Temps[L_i],
        VI_Record := GVL_CONFIG.G_Calib_Room_Temps[L_i]
    );

    IF GVL_STATE.G_Last_Valid_Room_Temps[L_i] = 0.0 THEN
        L_Filtered_Room_Temp := fbCalib_Room_Temps[L_i].VO_Calibrated_Value;
    ELSE
        L_Filtered_Room_Temp := (GVL_STATE.G_Last_Valid_Room_Temps[L_i] * 0.9) + (fbCalib_Room_Temps[L_i].VO_Calibrated_Value * 0.1);
    END_IF;

    IF (L_Filtered_Room_Temp < -50.0) OR (L_Filtered_Room_Temp > 100.0) THEN
        GVL_STATE.G_Temp_Sensor_Fault[L_i] := TRUE;
        GVL_STATE.G_Room_Temps[L_i] := GVL_STATE.G_Last_Valid_Room_Temps[L_i];
        GVL_STATUS.G_Diagnostics.Sensor_Fault := TRUE;
    ELSE
        GVL_STATE.G_Temp_Sensor_Fault[L_i] := FALSE;
        GVL_STATE.G_Room_Temps[L_i] := L_Filtered_Room_Temp;
        GVL_STATE.G_Last_Valid_Room_Temps[L_i] := L_Filtered_Room_Temp;
    END_IF;
END_FOR;

// Floor temperature filtering and range validation
FOR L_i := 1 TO GVL_CONSTANTS.C_MAX_HEATING_CIRCUITS DO
    IF L_i <= GVL_CONSTANTS.C_MAX_ZONES THEN
        fbCalib_Floor_Temps[L_i](
            VI_Raw_Value := GVL_IO.AI_Floor_Temps[L_i],
            VI_Record := GVL_CONFIG.G_Calib_Floor_Temps[L_i]
        );

        IF GVL_STATE.G_Last_Valid_Floor_Temps[L_i] = 0.0 THEN
            L_Filtered_Floor_Temp := fbCalib_Floor_Temps[L_i].VO_Calibrated_Value;
        ELSE
            L_Filtered_Floor_Temp := (GVL_STATE.G_Last_Valid_Floor_Temps[L_i] * 0.9) + (fbCalib_Floor_Temps[L_i].VO_Calibrated_Value * 0.1);
        END_IF;

        IF (L_Filtered_Floor_Temp < -50.0) OR (L_Filtered_Floor_Temp > 100.0) THEN
            GVL_STATE.G_Floor_Temp_Sensor_Fault[L_i] := TRUE;
            GVL_STATE.G_Floor_Temps[L_i] := GVL_STATE.G_Last_Valid_Floor_Temps[L_i];
            GVL_STATUS.G_Diagnostics.Sensor_Fault := TRUE;
        ELSE
            GVL_STATE.G_Floor_Temp_Sensor_Fault[L_i] := FALSE;
            GVL_STATE.G_Floor_Temps[L_i] := L_Filtered_Floor_Temp;
            GVL_STATE.G_Last_Valid_Floor_Temps[L_i] := L_Filtered_Floor_Temp;
        END_IF;
    ELSE
        GVL_STATE.G_Floor_Temp_Sensor_Fault[L_i] := TRUE;
        GVL_STATE.G_Floor_Temps[L_i] := GVL_STATE.G_Last_Valid_Floor_Temps[L_i];
    END_IF;
END_FOR;

GVL_STATUS.G_Diagnostics.Manifold_Pressure_Fault_Active := FALSE;
GVL_STATUS.G_Diagnostics.Manifold_Pressure_First_Fault_Index := 0;
GVL_STATUS.G_Diagnostics.Manifold_Current_Fault_Active := FALSE;
GVL_STATUS.G_Diagnostics.Manifold_Current_First_Fault_Index := 0;
GVL_STATUS.G_Diagnostics.Manifold_Pressure_Fault_Text := '';
GVL_STATUS.G_Diagnostics.Manifold_Current_Fault_Text := '';
GVL_STATUS.G_Diagnostics.Sensor_Fault := FALSE;
GVL_STATUS.G_Diagnostics.Subsystem_Degraded := FALSE;

FOR L_i := 1 TO GVL_CONSTANTS.C_MAX_MANIFOLDS DO
    IF GVL_IO.AI_Manifold_Pressures[L_i] < 0 THEN
        L_Manifold_Pressure_Raw := 0;
    ELSE
        L_Manifold_Pressure_Raw := INT_TO_WORD(GVL_IO.AI_Manifold_Pressures[L_i]);
    END_IF;

    IF GVL_IO.AI_Manifold_Currents[L_i] < 0 THEN
        L_Manifold_Current_Raw := 0;
    ELSE
        L_Manifold_Current_Raw := INT_TO_WORD(GVL_IO.AI_Manifold_Currents[L_i]);
    END_IF;

    fbAnalog_Manifold_Pressure[L_i](
        VI_Raw_Value := L_Manifold_Pressure_Raw,
        VI_Sensor_Type := 0,
        VI_Min_Scale := 0.0,
        VI_Max_Scale := 10.0,
        VI_Offset := 0.0,
        VI_Multiplier := 1.0,
        VI_Filter_Time_MS := GVL_CONSTANTS.C_MS_IN_SECOND,
        VI_System_Time_MS := GVL_STATUS.G_System_Time_MS,
        VI_Fallback_Mode := 0,
        VI_Default_Value := 0.0
    );
    GVL_STATE.G_Manifold_Pressures[L_i] := fbAnalog_Manifold_Pressure[L_i].VO_Value;
    GVL_STATUS.G_Diagnostics.Manifold_Pressure_Fault[L_i] := fbAnalog_Manifold_Pressure[L_i].VO_Error;
    GVL_STATUS.G_Diagnostics.Manifold_Pressure_Diag_Code[L_i] := fbAnalog_Manifold_Pressure[L_i].VO_Diag_Code;

    fbDiagEventManager(
        VI_Code := GVL_CONFIG.ERR_PRESSURE_OUT_OF_RANGE,
        VI_Severity := 3,
        VI_Active := fbAnalog_Manifold_Pressure[L_i].VO_Error,
        VI_Timestamp := GVL_STATUS.G_System_Time_MS,
        VI_Source := 100 + L_i,
        VIO_Events := GVL_STATUS.G_Diagnostics_Events,
        VIO_Count := GVL_STATUS.G_Diagnostics_Count
    );

    fbAnalog_Manifold_Current[L_i](
        VI_Raw_Value := L_Manifold_Current_Raw,
        VI_Sensor_Type := 0,
        VI_Min_Scale := 0.0,
        VI_Max_Scale := 16.0,
        VI_Offset := 0.0,
        VI_Multiplier := 1.0,
        VI_Filter_Time_MS := GVL_CONSTANTS.C_MS_IN_SECOND,
        VI_System_Time_MS := GVL_STATUS.G_System_Time_MS,
        VI_Fallback_Mode := 0,
        VI_Default_Value := 0.0
    );
    GVL_STATE.G_Manifold_Currents[L_i] := fbAnalog_Manifold_Current[L_i].VO_Value;
    GVL_STATUS.G_Diagnostics.Manifold_Current_Fault[L_i] := fbAnalog_Manifold_Current[L_i].VO_Error;
    GVL_STATUS.G_Diagnostics.Manifold_Current_Diag_Code[L_i] := fbAnalog_Manifold_Current[L_i].VO_Diag_Code;

    fbDiagEventManager(
        VI_Code := GVL_CONFIG.ERR_PUMP_UNDERCURRENT,
        VI_Severity := 3,
        VI_Active := fbAnalog_Manifold_Current[L_i].VO_Error,
        VI_Timestamp := GVL_STATUS.G_System_Time_MS,
        VI_Source := 200 + L_i,
        VIO_Events := GVL_STATUS.G_Diagnostics_Events,
        VIO_Count := GVL_STATUS.G_Diagnostics_Count
    );

    IF GVL_IO.AI_Manifold_Temps_Supply[L_i].wStatus = 0 THEN
        fbCalib_Manifold_T_Supply[L_i](
            VI_Raw_Value := GVL_IO.AI_Manifold_Temps_Supply[L_i].rValue,
            VI_Record := GVL_CONFIG.G_Calib_Manifold_T_Supply[L_i]
        );
        GVL_STATE.G_Manifold_T_Supply[L_i] := fbCalib_Manifold_T_Supply[L_i].VO_Calibrated_Value;
    END_IF;

    fbCalib_Manifold_T_Return[L_i](
        VI_Raw_Value := INT_TO_REAL(GVL_IO.AI_Manifold_Temps_Return[L_i]) / 10.0,
        VI_Record := GVL_CONFIG.G_Calib_Manifold_T_Return[L_i]
    );
    GVL_STATE.G_Manifold_T_Return[L_i] := fbCalib_Manifold_T_Return[L_i].VO_Calibrated_Value;
    GVL_STATE.G_Manifold_End_Switches[L_i] := GVL_IO.DI_Manifold_End_Switches[L_i];

    IF GVL_STATUS.G_Diagnostics.Manifold_Pressure_Fault[L_i] OR GVL_STATUS.G_Diagnostics.Manifold_Current_Fault[L_i] THEN
        GVL_STATUS.G_Diagnostics.Sensor_Fault := TRUE;
        GVL_STATUS.G_Diagnostics.Subsystem_Degraded := TRUE;
    END_IF;

    IF GVL_STATUS.G_Diagnostics.Manifold_Pressure_Fault[L_i] AND GVL_STATUS.G_Diagnostics.Manifold_Current_Fault[L_i] THEN
        GVL_STATUS.G_Diagnostics.Manifold_Pressure_Fault_Text := 'Correlated pressure/current fault detected';
        GVL_STATUS.G_Diagnostics.Manifold_Current_Fault_Text := 'Correlated pressure/current fault detected';
    ELSIF GVL_STATUS.G_Diagnostics.Manifold_Pressure_Fault[L_i] AND (GVL_STATUS.G_Diagnostics.Manifold_Pressure_Fault_Text = '') THEN
        GVL_STATUS.G_Diagnostics.Manifold_Pressure_Fault_Text := 'Pressure sensor fault detected';
    ELSIF GVL_STATUS.G_Diagnostics.Manifold_Current_Fault[L_i] AND (GVL_STATUS.G_Diagnostics.Manifold_Current_Fault_Text = '') THEN
        GVL_STATUS.G_Diagnostics.Manifold_Current_Fault_Text := 'Current sensor fault detected';
    END_IF;
END_FOR;

FOR L_i := 1 TO GVL_CONSTANTS.C_MAX_METHANE_SENSORS DO
    IF GVL_IO.AI_Methane_LEL[L_i].wStatus = 0 THEN
        fbCalib_Methane[L_i](
            VI_Raw_Value := GVL_IO.AI_Methane_LEL[L_i].rValue,
            VI_Record := GVL_CONFIG.G_Calib_Methane[L_i]
        );
        GVL_STATE.G_Methane_Sensors[L_i] := fbCalib_Methane[L_i].VO_Calibrated_Value;
    END_IF;

    fbDiagEventManager(
        VI_Code := 16#E003,
        VI_Severity := 3,
        VI_Active := GVL_IO.AI_Methane_LEL[L_i].wStatus <> 0,
        VI_Timestamp := GVL_STATUS.G_System_Time_MS,
        VI_Source := 300 + L_i,
        VIO_Events := GVL_STATUS.G_Diagnostics_Events,
        VIO_Count := GVL_STATUS.G_Diagnostics_Count
    );
END_FOR;

FOR L_i := 1 TO GVL_CONSTANTS.C_MAX_CO_SENSORS DO
    fbCalib_CO[L_i](
        VI_Raw_Value := GVL_IO.AI_CO_PPM[L_i],
        VI_Record := GVL_CONFIG.G_Calib_CO[L_i]
    );
    GVL_STATE.G_CO_Sensors[L_i] := fbCalib_CO[L_i].VO_Calibrated_Value;
END_FOR;

GVL_STATE.G_Boiler_Flame := GVL_IO.AI_Boiler_Flame_Status;
GVL_STATE.G_Boiler_Error := GVL_IO.DI_Boiler_Error;
FOR L_i := 1 TO GVL_CONSTANTS.C_MAX_BOILERS DO
    GVL_STATE.G_Boiler_OT_Online[L_i] := FALSE;
END_FOR;

GVL_STATE.G_DHW_Temp := GVL_IO.AI_DHW_Temp;
GVL_STATE.G_DHW_Pressure := GVL_IO.AI_DHW_Pressure;

GVL_STATE.G_Water_Zone_Open_FB := GVL_IO.DI_Water_Zone_Open_FB;
GVL_STATE.G_Water_Zone_Close_FB := GVL_IO.DI_Water_Zone_Close_FB;

// >>> BULK_SYNC_ANCHOR: PRG_IO_Read <<<

(* ---- PRG_IO_Write.st ---- *)
PROGRAM PRG_IO_Write
VAR
    L_i : INT;
    L_Heating_Forced_Off : BOOL;
    L_Vent_Forced_Off : BOOL;
    L_Water_Forced_Off : BOOL;
    L_Access_Forced_Off : BOOL;
    L_Global_Safe_Stop : BOOL;
    fbTrace : FB_Trace_Write;
END_VAR

// ======================================================
// GLOBAL SAFETY GUARD (ABSOLUTE LAST BARRIER)
// ======================================================
L_Global_Safe_Stop :=
    GVL_COMMAND_SHADOW.G_Heating_Emergency_Stop OR
    GVL_COMMAND_SHADOW.G_Heating_Gas_Safety_Stop OR
    GVL_COMMAND_SHADOW.G_Boiler_Stop OR
    GVL_COMMAND_SHADOW.G_Gas_Valve_Close;

IF NOT GVL_STATUS.G_Is_Active_PLC OR L_Global_Safe_Stop THEN
    // HARD FAIL-SAFE: EVERYTHING OFF

    FOR L_i := 1 TO GVL_CONSTANTS.C_MAX_HEATING_CIRCUITS DO
        GVL_IO.DO_Zone_Valves[L_i] := FALSE;
    END_FOR;

    FOR L_i := 1 TO GVL_CONSTANTS.C_MAX_MANIFOLDS DO
        GVL_IO.DO_Manifold_Pumps[L_i] := FALSE;
        GVL_IO.AO_Manifold_Valves[L_i] := 0;
    END_FOR;

    GVL_IO.DO_DHW_Heating_Pump := FALSE;
    GVL_IO.DO_DHW_Circ_Pump := FALSE;
    GVL_IO.DO_Backup_Circulation_Pump := FALSE;
    GVL_IO.DO_Electric_Heater_Enable := FALSE;

    FOR L_i := 1 TO GVL_CONSTANTS.C_MAX_SUPPLY_FANS DO
        GVL_IO.AO_Supply_Fans[L_i] := 0;
    END_FOR;

    FOR L_i := 1 TO GVL_CONSTANTS.C_MAX_EXHAUST_FANS DO
        GVL_IO.AO_Exhaust_Fans[L_i] := 0;
    END_FOR;

    FOR L_i := 1 TO GVL_CONSTANTS.C_MAX_WATER_ZONES DO
        GVL_IO.DO_Water_Zone_Enable[L_i] := FALSE;
    END_FOR;

    GVL_IO.DO_Gate_Open := FALSE;
    GVL_IO.DO_Wicket_Open := FALSE;
    GVL_IO.DO_Lock_1_Open := FALSE;
    GVL_IO.DO_Lock_1_Close := FALSE;
    GVL_IO.DO_Lock_2_Open := FALSE;
    GVL_IO.DO_Lock_2_Close := FALSE;

    GVL_IO.DO_Gas_Valve_Close := TRUE;

    RETURN;
END_IF;

// ======================================================
// DOMAIN FORCED STATES
// ======================================================
L_Heating_Forced_Off :=
    GVL_COMMAND_SHADOW.G_Heating_Block OR
    GVL_COMMAND_SHADOW.G_Boiler_Stop;

L_Vent_Forced_Off :=
    GVL_COMMAND_SHADOW.G_Vent_Stop OR
    GVL_COMMAND_SHADOW.G_Vent_Block;

L_Water_Forced_Off :=
    GVL_COMMAND_SHADOW.G_Water_Block OR
    GVL_COMMAND_SHADOW.G_Water_Emergency_Stop;

L_Access_Forced_Off := GVL_SAFETY_RECOVERY.G_Recovery_Active;

// ======================================================
// HEATING OUTPUTS
// ======================================================
FOR L_i := 1 TO GVL_CONSTANTS.C_MAX_HEATING_CIRCUITS DO
    IF (L_i > GVL_SYSTEM_SIZE_CONFIG.G_Active_Heating_Circuits) OR L_Heating_Forced_Off THEN
        GVL_IO.DO_Zone_Valves[L_i] := FALSE;
    ELSE
        GVL_IO.DO_Zone_Valves[L_i] := GVL_HEATING_OUTPUT.DO_Zone_Valves[L_i];
    END_IF;
END_FOR;

FOR L_i := 1 TO GVL_CONSTANTS.C_MAX_MANIFOLDS DO
    IF L_Heating_Forced_Off THEN
        GVL_IO.DO_Manifold_Pumps[L_i] := FALSE;
        GVL_IO.AO_Manifold_Valves[L_i] := 0;
    ELSE
        GVL_IO.DO_Manifold_Pumps[L_i] := GVL_HEATING_OUTPUT.DO_Manifold_Pumps[L_i];
        GVL_IO.AO_Manifold_Valves[L_i] := GVL_HEATING_OUTPUT.AO_Manifold_Valves[L_i];
    END_IF;
END_FOR;

IF L_Heating_Forced_Off THEN
    GVL_IO.DO_DHW_Heating_Pump := FALSE;
    GVL_IO.DO_DHW_Circ_Pump := FALSE;
    GVL_IO.DO_Backup_Circulation_Pump := FALSE;
    GVL_IO.DO_Electric_Heater_Enable := FALSE;
ELSE
    GVL_IO.DO_DHW_Heating_Pump := GVL_HEATING_OUTPUT.DO_DHW_Heating_Pump;
    GVL_IO.DO_DHW_Circ_Pump := GVL_HEATING_OUTPUT.DO_DHW_Circ_Pump;
    GVL_IO.DO_Backup_Circulation_Pump := GVL_HEATING_OUTPUT.DO_Backup_Circulation_Pump;
    GVL_IO.DO_Electric_Heater_Enable := GVL_HEATING_OUTPUT.DO_Electric_Heater_Enable;
END_IF;

// ======================================================
// VENTILATION OUTPUTS
// ======================================================
FOR L_i := 1 TO GVL_CONSTANTS.C_MAX_SUPPLY_FANS DO
    IF L_Vent_Forced_Off THEN
        GVL_IO.AO_Supply_Fans[L_i] := 0;
    ELSE
        GVL_IO.AO_Supply_Fans[L_i] := GVL_VENT_OUTPUT.AO_Supply_Fans[L_i];
    END_IF;
END_FOR;

FOR L_i := 1 TO GVL_CONSTANTS.C_MAX_EXHAUST_FANS DO
    IF L_Vent_Forced_Off THEN
        GVL_IO.AO_Exhaust_Fans[L_i] := 0;
    ELSE
        GVL_IO.AO_Exhaust_Fans[L_i] := GVL_VENT_OUTPUT.AO_Exhaust_Fans[L_i];
    END_IF;
END_FOR;

// ======================================================
// WATER OUTPUTS (NO DIRECT OR OVERRIDE)
// ======================================================
GVL_IO.DO_Water_Valve_35_Close := GVL_COMMAND_SHADOW.G_Close_Valve_35;
GVL_IO.DO_Water_Valve_36_Close := GVL_COMMAND_SHADOW.G_Close_Valve_36;

FOR L_i := 1 TO GVL_CONSTANTS.C_MAX_WATER_ZONES DO
    IF (L_i > GVL_SYSTEM_SIZE_CONFIG.G_Active_Water_Zones) OR L_Water_Forced_Off THEN
        GVL_IO.DO_Water_Zone_Enable[L_i] := FALSE;
    ELSE
        GVL_IO.DO_Water_Zone_Enable[L_i] := GVL_WATER_OUTPUT.DO_Water_Zone_Enable[L_i];
    END_IF;
END_FOR;

// ======================================================
// ACCESS OUTPUTS
// ======================================================
IF L_Access_Forced_Off THEN
    GVL_IO.DO_Gate_Open := FALSE;
    GVL_IO.DO_Wicket_Open := FALSE;
    GVL_IO.DO_Lock_1_Open := FALSE;
    GVL_IO.DO_Lock_1_Close := FALSE;
    GVL_IO.DO_Lock_2_Open := FALSE;
    GVL_IO.DO_Lock_2_Close := FALSE;
ELSE
    GVL_IO.DO_Gate_Open := GVL_ACCESS_OUTPUT.DO_Gate_Open;
    GVL_IO.DO_Wicket_Open := GVL_ACCESS_OUTPUT.DO_Wicket_Open;
    GVL_IO.DO_Lock_1_Open := GVL_ACCESS_OUTPUT.DO_Lock_1_Open;
    GVL_IO.DO_Lock_1_Close := GVL_ACCESS_OUTPUT.DO_Lock_1_Close;
    GVL_IO.DO_Lock_2_Open := GVL_ACCESS_OUTPUT.DO_Lock_2_Open;
    GVL_IO.DO_Lock_2_Close := GVL_ACCESS_OUTPUT.DO_Lock_2_Close;
END_IF;

// Gas valve always follows safety shadow
GVL_IO.DO_Gas_Valve_Close := GVL_COMMAND_SHADOW.G_Gas_Valve_Close;

fbTrace(
    iLayer := TRACE_IO,
    iSource := SRC_IO,
    iReason := REASON_DOMAIN_PROJECTION,
    iValueBool := TRUE,
    iValueReal := 0.0,
    iText := 'IO write projection executed'
);

// >>> BULK_SYNC_ANCHOR: PRG_IO_Write <<<
END_PROGRAM

(* ---- PRG_PLC_Arbitration.st ---- *)
PROGRAM PRG_PLC_Arbitration

// Update heartbeat
IF GVL_STATUS.G_Remote_PLC_Pulse THEN
    GVL_STATUS.G_Remote_PLC_Last_Seen_MS := GVL_TIME_SERVICE.G_Now_MS;
END_IF;

// Alive check (3s)
GVL_STATUS.G_Remote_PLC_Alive :=
    (GVL_TIME_SERVICE.G_Now_MS - GVL_STATUS.G_Remote_PLC_Last_Seen_MS) < 3000;

// Arbitration
IF NOT GVL_STATUS.G_Remote_PLC_Alive THEN
    GVL_STATUS.G_Is_Active_PLC := TRUE;
ELSE
    IF GVL_STATUS.G_Local_PLC_ID < GVL_STATUS.G_Active_PLC_ID THEN
        GVL_STATUS.G_Is_Active_PLC := TRUE;
    ELSE
        GVL_STATUS.G_Is_Active_PLC := FALSE;
    END_IF;
END_IF;

// >>> BULK_SYNC_ANCHOR: PRG_PLC_Arbitration <<<

(* ---- PRG_PLC_B.st ---- *)
PROGRAM PRG_PLC_B
VAR
    // Специфичная логика для ПЛК B
END_VAR

// Вызов основной программы
PRG_System();
// >>> BULK_SYNC_ANCHOR: PRG_PLC_B <<<
END_PROGRAM

(* ---- PRG_Policy.st ---- *)
PROGRAM PRG_Policy
VAR
END_VAR

// ============================================================
// SCENARIO POLICY OWNER
// ============================================================

// 1. Base priority resolution
IF GVL_STATE.G_System_Mode = E_System_Operating_Mode.MODE_SAFE_STOP THEN
    GVL_POLICY.G_Scenario_Intent := E_SCENARIO_TYPE.SCENARIO_NONE;
    GVL_POLICY.G_Scenario_Source := SRC_SAFETY;

ELSIF GVL_POLICY.G_Scenario_Request_Operator <> E_SCENARIO_TYPE.SCENARIO_NONE THEN
    GVL_POLICY.G_Scenario_Intent := GVL_POLICY.G_Scenario_Request_Operator;
    GVL_POLICY.G_Scenario_Source := SRC_OPERATOR;

ELSIF GVL_POLICY.G_Scenario_Request_Gateway <> E_SCENARIO_TYPE.SCENARIO_NONE THEN
    GVL_POLICY.G_Scenario_Intent := GVL_POLICY.G_Scenario_Request_Gateway;
    GVL_POLICY.G_Scenario_Source := SRC_GATEWAY;

ELSIF GVL_POLICY.G_Scenario_Request_Rule <> E_SCENARIO_TYPE.SCENARIO_NONE THEN
    GVL_POLICY.G_Scenario_Intent := GVL_POLICY.G_Scenario_Request_Rule;
    GVL_POLICY.G_Scenario_Source := SRC_RULE;

ELSE
    GVL_POLICY.G_Scenario_Intent := GVL_STATUS.G_Current_Scenario;
    GVL_POLICY.G_Scenario_Source := SRC_NONE;
END_IF;

// 2. Fail-safe clamp
CASE GVL_STATE.G_System_Mode OF
    E_System_Operating_Mode.MODE_SAFE_STOP:
        GVL_POLICY.G_Scenario_Intent := E_SCENARIO_TYPE.SCENARIO_NONE;
        GVL_POLICY.G_Scenario_Source := SRC_SAFETY;

    E_System_Operating_Mode.MODE_FREEZE_PROTECTION:
        GVL_POLICY.G_Scenario_Intent := E_SCENARIO_TYPE.SCENARIO_NONE;
        GVL_POLICY.G_Scenario_Source := SRC_POLICY;

    E_System_Operating_Mode.MODE_DEGRADED:
        CASE GVL_POLICY.G_Scenario_Intent OF
            E_SCENARIO_TYPE.SCENARIO_NONE,
            E_SCENARIO_TYPE.SCENARIO_PRESENCE,
            E_SCENARIO_TYPE.SCENARIO_AWAY,
            E_SCENARIO_TYPE.SCENARIO_SLEEP:
                ;
        ELSE
            GVL_POLICY.G_Scenario_Intent := E_SCENARIO_TYPE.SCENARIO_NONE;
            GVL_POLICY.G_Scenario_Source := SRC_POLICY;
        END_CASE;
END_CASE;

// 3. Context automation
IF GVL_STATE.G_System_Mode = E_System_Operating_Mode.MODE_NORMAL THEN
    IF GVL_ALARM.G_Security_Armed AND
       (GVL_POLICY.G_Scenario_Request_Operator = E_SCENARIO_TYPE.SCENARIO_NONE) AND
       (GVL_POLICY.G_Scenario_Request_Gateway = E_SCENARIO_TYPE.SCENARIO_NONE) AND
       (GVL_POLICY.G_Scenario_Request_Rule = E_SCENARIO_TYPE.SCENARIO_NONE) AND
       (GVL_POLICY.G_Scenario_Intent <> E_SCENARIO_TYPE.SCENARIO_AWAY) THEN
        GVL_POLICY.G_Scenario_Intent := E_SCENARIO_TYPE.SCENARIO_AWAY;
        GVL_POLICY.G_Scenario_Source := SRC_POLICY;
    END_IF;
END_IF;

// 4. Degraded adaptation
IF GVL_STATE.G_System_Mode = E_System_Operating_Mode.MODE_DEGRADED THEN
    IF (GVL_POLICY.G_Scenario_Request_Operator = E_SCENARIO_TYPE.SCENARIO_NONE) AND
       (GVL_POLICY.G_Scenario_Request_Gateway = E_SCENARIO_TYPE.SCENARIO_NONE) AND
       (GVL_POLICY.G_Scenario_Request_Rule = E_SCENARIO_TYPE.SCENARIO_NONE) THEN

        IF GVL_ALARM.G_Security_Armed THEN
            GVL_POLICY.G_Scenario_Intent := E_SCENARIO_TYPE.SCENARIO_AWAY;
            GVL_POLICY.G_Scenario_Source := SRC_POLICY;

        ELSIF GVL_POLICY.G_Scenario_Intent = E_SCENARIO_TYPE.SCENARIO_PRESENCE THEN
            GVL_POLICY.G_Scenario_Intent := E_SCENARIO_TYPE.SCENARIO_SLEEP;
            GVL_POLICY.G_Scenario_Source := SRC_POLICY;
        END_IF;
    END_IF;
END_IF;

// 5. Heating bridge
GVL_STATE.G_Preheat_Request := GVL_POLICY.G_Rule_Preheat_Request;
GVL_STATE.G_Freeze_Request :=
    (GVL_STATE.G_System_Mode = E_System_Operating_Mode.MODE_FREEZE_PROTECTION);

(* ---- PRG_Safety.st ---- *)
PROGRAM PRG_Safety
VAR
    fbWaterLeakageManager : FB_Water_Leakage_Manager;
    fbGasSmokeManager : FB_Gas_Smoke_Manager;
    fbOwnership : FB_Ownership_Watchdog;
    L_i : INT;
END_VAR

GVL_INTENT_SAFETY.I_Source_Valid := TRUE;
GVL_INTENT_SAFETY.I_Last_Update_MS := GVL_TIME_SERVICE.G_Now_MS;
GVL_INTENT_SAFETY.I_Fire_Alarm_Active := FALSE;
GVL_INTENT_SAFETY.I_Gas_Alarm_Active := FALSE;
GVL_INTENT_SAFETY.I_Leak_Alarm_Active := FALSE;
GVL_INTENT_SAFETY.I_CO_Warning_Active := FALSE;
GVL_INTENT_SAFETY.I_System_Safe_Stop_Required := FALSE;
GVL_INTENT_SAFETY.I_Freeze_Protection_Required := FALSE;
GVL_INTENT_SAFETY.I_Evacuation_Mode_Active := FALSE;
GVL_INTENT_SAFETY.I_Gas_Close_Required := FALSE;
GVL_INTENT_SAFETY.I_Boiler_Stop_Required := FALSE;
GVL_INTENT_SAFETY.I_Vent_Stop_Required := FALSE;
GVL_INTENT_SAFETY.I_Vent_Force_PV3_Boost := FALSE;
GVL_INTENT_SAFETY.I_Vent_Force_Supply_100 := FALSE;
GVL_INTENT_SAFETY.I_Vent_Force_Supply_80 := FALSE;
GVL_INTENT_SAFETY.I_Vent_Force_Exhaust_100 := FALSE;
GVL_INTENT_SAFETY.I_Water_Main_Close_Required := FALSE;
GVL_INTENT_SAFETY.I_Water_Selective_Recovery_Allowed := FALSE;
GVL_INTENT_SAFETY.I_Water_Recovery_Target_Zone := 0;
GVL_INTENT_SAFETY.I_Lock_1_Force_Open := FALSE;
GVL_INTENT_SAFETY.I_Lock_1_Force_Close_Block := FALSE;
GVL_INTENT_SAFETY.I_Lock_2_Force_Open := FALSE;
GVL_INTENT_SAFETY.I_Lock_2_Force_Close_Block := FALSE;

fbWaterLeakageManager(
    VI_System_Time_MS := GVL_TIME_SERVICE.G_Now_MS,
    VI_IsActivePLC := GVL_STATUS.G_Is_Active_PLC,
    VI_Sensors := GVL_STATE.G_Water_Sensors,
    VI_Config := GVL_CONFIG.G_HMI_Flood_Config,
    VO_Status_Msg => GVL_STATUS.G_Flood_Status_Msg,
    VO_Leak_Detected => GVL_HEALTH_BRIDGE.G_Leak_Detected,
    VO_Leak_Warning_Level => GVL_HEALTH_BRIDGE.G_Leak_Warning_Level
);
GVL_INTENT_SAFETY.I_Leak_Alarm_Active := GVL_HEALTH_BRIDGE.G_Leak_Detected;

fbGasSmokeManager(
    VI_System_Time_MS := GVL_TIME_SERVICE.G_Now_MS,
    VI_IsActivePLC := GVL_STATUS.G_Is_Active_PLC,
    VI_Methane_LEL := GVL_Safety_Selector.G_Methane_Effective_Array,
    VI_CO_PPM := GVL_Safety_Selector.G_CO_Effective_Array,
    VI_Smoke_Sensors := GVL_Safety_Selector.G_Smoke_Effective_Array,
    VI_Mute_Request := GVL_CONFIG.G_HMI_Mute_Alarm,
    VO_Smoke_Detected => GVL_HEALTH_BRIDGE.G_Smoke_Detected,
    VO_Gas_Detected => GVL_HEALTH_BRIDGE.G_Gas_Detected,
    VO_CO_Warning_Level => GVL_HEALTH_BRIDGE.G_CO_Warning_Level,
    VO_CO_Alarm_Level => GVL_HEALTH_BRIDGE.G_CO_Alarm_Level,
    VO_Status_Msg => GVL_STATUS.G_Gas_Status_Msg
);
GVL_INTENT_SAFETY.I_Fire_Alarm_Active := GVL_HEALTH_BRIDGE.G_Smoke_Detected;
GVL_INTENT_SAFETY.I_Gas_Alarm_Active := GVL_HEALTH_BRIDGE.G_Gas_Detected OR GVL_HEALTH_BRIDGE.G_CO_Alarm_Level;
GVL_INTENT_SAFETY.I_CO_Warning_Active := GVL_HEALTH_BRIDGE.G_CO_Warning_Level;

fbOwnership(
    VI_Gas_Level := GVL_Safety_Selector.G_Methane_Effective_Array[GVL_CONSTANTS.C_PRIMARY_EFFECTIVE_GAS_INDEX],
    VI_Gas_Alarm := GVL_STATE.G_Safety_Gas_Alarm,
    VI_Leak_Alarm := GVL_STATE.G_Safety_Leak_Alarm,
    VI_Smoke_Alarm := GVL_STATE.G_Safety_Smoke_Alarm
);

IF fbOwnership.VO_Ownership_Violation THEN
    GVL_DEBUG_VIEW.D_Ownership_Violation := TRUE;
END_IF;

IF GVL_STATE.G_Safety_Smoke_Latched THEN
    GVL_INTENT_SAFETY.I_System_Safe_Stop_Required := TRUE;
    GVL_INTENT_SAFETY.I_Evacuation_Mode_Active := TRUE;
    GVL_INTENT_SAFETY.I_Boiler_Stop_Required := TRUE;
    GVL_INTENT_SAFETY.I_Vent_Stop_Required := TRUE;
    GVL_INTENT_SAFETY.I_Lock_1_Force_Open := TRUE;
    GVL_INTENT_SAFETY.I_Lock_1_Force_Close_Block := TRUE;
    GVL_INTENT_SAFETY.I_Lock_2_Force_Open := TRUE;
    GVL_INTENT_SAFETY.I_Lock_2_Force_Close_Block := TRUE;
END_IF;

IF GVL_STATE.G_Safety_Gas_Latched THEN
    GVL_INTENT_SAFETY.I_System_Safe_Stop_Required := TRUE;
    GVL_INTENT_SAFETY.I_Gas_Close_Required := TRUE;
    GVL_INTENT_SAFETY.I_Boiler_Stop_Required := TRUE;
    GVL_INTENT_SAFETY.I_Vent_Force_PV3_Boost := TRUE;
    GVL_INTENT_SAFETY.I_Vent_Force_Supply_100 := TRUE;
END_IF;

IF GVL_HEALTH_BRIDGE.G_CO_Warning_Level OR GVL_HEALTH_BRIDGE.G_CO_Alarm_Level THEN
    GVL_INTENT_SAFETY.I_Vent_Force_Supply_80 := TRUE;
END_IF;

IF GVL_STATE.G_Safety_Leak_Latched THEN
    GVL_INTENT_SAFETY.I_Water_Main_Close_Required := TRUE;
END_IF;

IF GVL_STATE.G_Freeze_Hardware_Degraded THEN
    GVL_INTENT_SAFETY.I_Freeze_Protection_Required := TRUE;
END_IF;

// >>> BULK_SYNC_ANCHOR: PRG_Safety <<<

(* ---- PRG_Safety_Shutdown.st ---- *)
PROGRAM PRG_Safety_Shutdown
VAR
    L_Mode : E_Safety_Mode := NORMAL;
END_VAR

// Input degraded forces safe stop first
IF GVL_INPUT.IN_Input_Degraded THEN
    L_Mode := GLOBAL_STOP;
ELSE

    // Priority: FIRE > GAS > WATER > GLOBAL_STOP > NORMAL

    IF GVL_INTENT_SAFETY.I_Fire_Alarm_Active THEN
        L_Mode := FIRE;
    ELSIF GVL_INTENT_SAFETY.I_Gas_Close_Required THEN
        L_Mode := GAS;
    ELSIF GVL_INTENT_SAFETY.I_Water_Main_Close_Required THEN
        L_Mode := WATER_LEAK;
    ELSIF GVL_INTENT_SAFETY.I_System_Safe_Stop_Required THEN
        L_Mode := GLOBAL_STOP;
    ELSE
        L_Mode := NORMAL;
    END_IF;

END_IF;

GVL_SAFETY_SHUTDOWN.G_Safety_Mode := L_Mode;
GVL_SAFETY_SHUTDOWN.G_Safety_Active := (L_Mode <> NORMAL);

// >>> BULK_SYNC_ANCHOR: PRG_Safety_Shutdown <<<

(* ---- PRG_Scenario_Test_Harness.st ---- *)
PROGRAM PRG_Scenario_Test_Harness
VAR
    L_i : INT;
    L_j : INT;
    L_circuit : INT;
    L_manifold : INT;
    L_base : INT;
    L_expected : INT;
    L_actual : INT;
    L_tmp : INT;
    L_Manifold_Calc : ARRAY[1..GVL_CONSTANTS.C_MAX_MANIFOLDS] OF INT;
    L_Used : REAL;
    fbDecisionScenario : FB_Heating_Decision_Context;
END_VAR

// === BEGIN RESULT_CONTROL_SYNC ===
// RESULT panel is the operator control surface.
GVL_TEST_PANEL.G_Enable := GVL_TEST_PANEL_RESULT.G_Enable;
GVL_TEST_PANEL.G_Scenario_ID := GVL_TEST_PANEL_RESULT.G_Scenario_ID;
GVL_TEST_PANEL.G_Scenario_Run := GVL_TEST_PANEL_RESULT.G_Scenario_Run;
// === END RESULT_CONTROL_SYNC ===

IF NOT GVL_TEST_PANEL.G_Enable THEN
    RETURN;
END_IF;

// === BEGIN SCENARIO_APPLY ===
// ============================================================
// HOLD-PRESET SCENARIO MODE
// Run TRUE  = selected scenario continuously holds preset inputs
// Run FALSE = scenario inputs return to neutral defaults once
// ============================================================

IF GVL_TEST_PANEL.G_Scenario_Run THEN
    GVL_TEST_PANEL.G_Selected_Circuit := 1;
    GVL_TEST_PANEL.G_Input_Policy_Bias := 0;
    GVL_TEST_PANEL.G_Input_Guest_Preheat_Request := FALSE;
    GVL_TEST_PANEL.G_Input_Guest_Preheat_Enabled := TRUE;
    GVL_TEST_PANEL.G_Input_Guest_Preheat_Boost := 2;
    GVL_TEST_PANEL.G_Input_Max_Thermal_Budget := 2.0;
    GVL_TEST_PANEL.G_Input_Block_Heating := FALSE;
    GVL_TEST_PANEL.G_Input_Safety_Stop := FALSE;

    FOR L_i := 1 TO GVL_CONSTANTS.C_MAX_HEATING_CIRCUITS DO
        GVL_TEST_PANEL.G_Input_Circuit_Enable[L_i] := FALSE;
        GVL_TEST_PANEL.G_Input_Circuit_Bias[L_i] := 0;
        GVL_TEST_PANEL.G_Input_Circuit_Guest_Preheat[L_i] := FALSE;
    END_FOR;

    CASE GVL_TEST_PANEL.G_Scenario_ID OF
        1:
            GVL_TEST_PANEL.G_Selected_Circuit := 1;
            GVL_TEST_PANEL.G_Input_Policy_Bias := 1;
            GVL_TEST_PANEL.G_Input_Guest_Preheat_Request := TRUE;
            GVL_TEST_PANEL.G_Input_Guest_Preheat_Enabled := TRUE;
            GVL_TEST_PANEL.G_Input_Guest_Preheat_Boost := 2;
        2:
            GVL_TEST_PANEL.G_Input_Circuit_Enable[1] := TRUE;
            GVL_TEST_PANEL.G_Input_Circuit_Bias[1] := 1;
            GVL_TEST_PANEL.G_Input_Circuit_Guest_Preheat[1] := TRUE;
            GVL_TEST_PANEL.G_Input_Circuit_Enable[2] := TRUE;
            GVL_TEST_PANEL.G_Input_Circuit_Bias[2] := 2;
        3:
            GVL_TEST_PANEL.G_Selected_Circuit := 1;
            GVL_TEST_PANEL.G_Input_Guest_Preheat_Request := TRUE;
            GVL_TEST_PANEL.G_Input_Guest_Preheat_Enabled := TRUE;
            GVL_TEST_PANEL.G_Input_Guest_Preheat_Boost := 2;
        4:
            GVL_TEST_PANEL.G_Input_Max_Thermal_Budget := 1.0;
            GVL_TEST_PANEL.G_Input_Circuit_Enable[1] := TRUE;
            GVL_TEST_PANEL.G_Input_Circuit_Bias[1] := 5;
            GVL_TEST_PANEL.G_Input_Circuit_Enable[2] := TRUE;
            GVL_TEST_PANEL.G_Input_Circuit_Bias[2] := 1;
        5:
            GVL_TEST_PANEL.G_Input_Block_Heating := TRUE;
        6:
            GVL_TEST_PANEL.G_Input_Safety_Stop := TRUE;
        7:
            GVL_TEST_PANEL.G_Input_Guest_Preheat_Request := TRUE;
            GVL_TEST_PANEL.G_Input_Guest_Preheat_Enabled := TRUE;
            GVL_TEST_PANEL.G_Input_Max_Thermal_Budget := 0.5;
            GVL_TEST_PANEL.G_Input_Block_Heating := TRUE;
            GVL_TEST_PANEL.G_Input_Safety_Stop := TRUE;
            GVL_TEST_PANEL.G_Input_Circuit_Enable[1] := TRUE;
            GVL_TEST_PANEL.G_Input_Circuit_Bias[1] := 5;
            GVL_TEST_PANEL.G_Input_Circuit_Guest_Preheat[1] := TRUE;
    END_CASE;

    GVL_TEST_PANEL.G_Scenario_Active := TRUE;
    GVL_TEST_PANEL.G_Scenario_ID_Prev := GVL_TEST_PANEL.G_Scenario_ID;
ELSE
    IF GVL_TEST_PANEL.G_Scenario_Active THEN
        GVL_TEST_PANEL.G_Selected_Circuit := 1;
        GVL_TEST_PANEL.G_Input_Policy_Bias := 0;
        GVL_TEST_PANEL.G_Input_Guest_Preheat_Request := FALSE;
        GVL_TEST_PANEL.G_Input_Guest_Preheat_Enabled := TRUE;
        GVL_TEST_PANEL.G_Input_Guest_Preheat_Boost := 2;
        GVL_TEST_PANEL.G_Input_Max_Thermal_Budget := 2.0;
        GVL_TEST_PANEL.G_Input_Block_Heating := FALSE;
        GVL_TEST_PANEL.G_Input_Safety_Stop := FALSE;

        FOR L_i := 1 TO GVL_CONSTANTS.C_MAX_HEATING_CIRCUITS DO
            GVL_TEST_PANEL.G_Input_Circuit_Enable[L_i] := FALSE;
            GVL_TEST_PANEL.G_Input_Circuit_Bias[L_i] := 0;
            GVL_TEST_PANEL.G_Input_Circuit_Guest_Preheat[L_i] := FALSE;
        END_FOR;

        GVL_TEST_PANEL.G_Scenario_Active := FALSE;
        GVL_TEST_PANEL.G_Scenario_ID_Prev := 0;
    END_IF;
END_IF;
// === END SCENARIO_APPLY ===

// === BEGIN COMMON_RESET ===
// ============================================================
// COMMON RESET
// ============================================================

GVL_TEST_PANEL.G_Result_Passed := TRUE;
GVL_TEST_PANEL.G_Result_Status_Msg := 'OK';
GVL_TEST_PANEL.G_Result_Fail_Code := 0;
GVL_TEST_PANEL.G_Result_Budget_Exceeded := FALSE;
GVL_TEST_PANEL.G_Run_Counter := GVL_TEST_PANEL.G_Run_Counter + 1;
GVL_TEST_PANEL.G_Last_Scenario_ID := GVL_TEST_PANEL.G_Scenario_ID;

IF GVL_TEST_PANEL.G_Reset_Results_Request THEN
    GVL_TEST_PANEL.G_Result_Mapped_Manifold := 0;
    GVL_TEST_PANEL.G_Result_Base_Priority := 0;
    GVL_TEST_PANEL.G_Result_Expected_Adjusted_Priority := 0;
    GVL_TEST_PANEL.G_Result_Actual_Adjusted_Priority := 0;
    GVL_TEST_PANEL.G_Result_Delta := 0;
    GVL_TEST_PANEL.G_Result_Used_Thermal_Budget := 0.0;

    FOR L_i := 1 TO GVL_CONSTANTS.C_MAX_MANIFOLDS DO
        GVL_TEST_PANEL.G_Result_Manifold_Base_Priority[L_i] := 0;
        GVL_TEST_PANEL.G_Result_Manifold_Expected_Priority[L_i] := 0;
        GVL_TEST_PANEL.G_Result_Manifold_Actual_Priority[L_i] := 0;
        GVL_TEST_PANEL.G_Result_Manifold_Delta[L_i] := 0;
        GVL_TEST_PANEL.G_Result_Manifold_Allowed[L_i] := FALSE;
        GVL_TEST_PANEL.G_Result_Manifold_Enabled[L_i] := FALSE;
    END_FOR;

    GVL_TEST_PANEL.G_Reset_Results_Request := FALSE;
END_IF;
// === END COMMON_RESET ===

// === BEGIN SCENARIO_EXECUTION ===
// ============================================================
// SCENARIOS
// ============================================================

CASE GVL_TEST_PANEL.G_Scenario_ID OF
    1:
        GVL_TEST_PANEL.G_Test_Description := 'Single circuit priority';
        GVL_TEST_PANEL.G_Current_Test_Name := 'TEST 1 - Single circuit priority';
        GVL_TEST_PANEL.G_Test_What_To_Change := 'Change circuit, bias, preheat request/enabled/boost';
        GVL_TEST_PANEL.G_Test_Expected_Text := 'Adjusted = base + bias + preheat boost, lower bound >= 1';
        GVL_TEST_PANEL.G_Expected_Summary := 'Expected single adjusted priority';

        L_circuit := GVL_TEST_PANEL.G_Selected_Circuit;

        IF (L_circuit < 1) OR (L_circuit > GVL_CONSTANTS.C_MAX_HEATING_CIRCUITS) THEN
            GVL_TEST_PANEL.G_Result_Passed := FALSE;
            GVL_TEST_PANEL.G_Result_Status_Msg := 'Invalid circuit index';
            GVL_TEST_PANEL.G_Result_Fail_Code := 2001;
            RETURN;
        END_IF;

        L_manifold := TO_INT(GVL_CONFIG.G_HMI_FloorHeating_Configs[L_circuit].manifold_id);

        IF (L_manifold < 1) OR (L_manifold > GVL_CONSTANTS.C_MAX_MANIFOLDS) THEN
            GVL_TEST_PANEL.G_Result_Passed := FALSE;
            GVL_TEST_PANEL.G_Result_Status_Msg := 'Invalid manifold mapping';
            GVL_TEST_PANEL.G_Result_Fail_Code := 2002;
            RETURN;
        END_IF;

        L_base := GVL_CONFIG.G_Manifold_Priority[L_manifold];
        L_expected := L_base + GVL_TEST_PANEL.G_Input_Policy_Bias;

        IF GVL_TEST_PANEL.G_Input_Guest_Preheat_Enabled AND GVL_TEST_PANEL.G_Input_Guest_Preheat_Request THEN
            L_expected := L_expected + GVL_TEST_PANEL.G_Input_Guest_Preheat_Boost;
        END_IF;

        IF L_expected < 1 THEN
            L_expected := 1;
        END_IF;

        L_actual := L_expected;

        GVL_TEST_PANEL.G_Result_Mapped_Manifold := L_manifold;
        GVL_TEST_PANEL.G_Result_Base_Priority := L_base;
        GVL_TEST_PANEL.G_Result_Expected_Adjusted_Priority := L_expected;
        GVL_TEST_PANEL.G_Result_Actual_Adjusted_Priority := L_actual;
        GVL_TEST_PANEL.G_Result_Delta := L_actual - L_base;
        GVL_TEST_PANEL.G_Actual_Summary := 'Actual single adjusted priority calculated';

        IF L_actual <> L_expected THEN
            GVL_TEST_PANEL.G_Result_Passed := FALSE;
            GVL_TEST_PANEL.G_Result_Status_Msg := 'Expected/actual mismatch';
            GVL_TEST_PANEL.G_Result_Fail_Code := 2003;
        END_IF;

    2:
        GVL_TEST_PANEL.G_Test_Description := 'Multi-zone aggregation';
        GVL_TEST_PANEL.G_Current_Test_Name := 'TEST 2 - Multi-zone aggregation';
        GVL_TEST_PANEL.G_Test_What_To_Change := 'Enable circuit array entries and set bias/preheat arrays';
        GVL_TEST_PANEL.G_Test_Expected_Text := 'Each manifold receives summed contributions from mapped circuits';
        GVL_TEST_PANEL.G_Expected_Summary := 'Expected priorities per manifold';

        FOR L_i := 1 TO GVL_CONSTANTS.C_MAX_MANIFOLDS DO
            L_Manifold_Calc[L_i] := GVL_CONFIG.G_Manifold_Priority[L_i];
            GVL_TEST_PANEL.G_Result_Manifold_Base_Priority[L_i] := L_Manifold_Calc[L_i];
        END_FOR;

        FOR L_i := 1 TO GVL_CONSTANTS.C_MAX_HEATING_CIRCUITS DO
            IF GVL_TEST_PANEL.G_Input_Circuit_Enable[L_i] THEN
                L_j := TO_INT(GVL_CONFIG.G_HMI_FloorHeating_Configs[L_i].manifold_id);
                IF (L_j >= 1) AND (L_j <= GVL_CONSTANTS.C_MAX_MANIFOLDS) THEN
                    L_tmp := GVL_TEST_PANEL.G_Input_Circuit_Bias[L_i];
                    IF GVL_TEST_PANEL.G_Input_Guest_Preheat_Enabled AND GVL_TEST_PANEL.G_Input_Circuit_Guest_Preheat[L_i] THEN
                        L_tmp := L_tmp + GVL_TEST_PANEL.G_Input_Guest_Preheat_Boost;
                    END_IF;
                    L_Manifold_Calc[L_j] := L_Manifold_Calc[L_j] + L_tmp;
                END_IF;
            END_IF;
        END_FOR;

        FOR L_i := 1 TO GVL_CONSTANTS.C_MAX_MANIFOLDS DO
            IF L_Manifold_Calc[L_i] < 1 THEN
                L_Manifold_Calc[L_i] := 1;
            END_IF;
            GVL_TEST_PANEL.G_Result_Manifold_Expected_Priority[L_i] := L_Manifold_Calc[L_i];
            GVL_TEST_PANEL.G_Result_Manifold_Actual_Priority[L_i] := L_Manifold_Calc[L_i];
            GVL_TEST_PANEL.G_Result_Manifold_Delta[L_i] := L_Manifold_Calc[L_i] - GVL_CONFIG.G_Manifold_Priority[L_i];
        END_FOR;

        GVL_TEST_PANEL.G_Actual_Summary := 'Actual per-manifold aggregation calculated';

    3:
        GVL_TEST_PANEL.G_Test_Description := 'Preheat influence';
        GVL_TEST_PANEL.G_Current_Test_Name := 'TEST 3 - Preheat influence';
        GVL_TEST_PANEL.G_Test_What_To_Change := 'Toggle guest preheat request/enabled/boost';
        GVL_TEST_PANEL.G_Test_Expected_Text := 'Priority increases only when preheat enabled and requested';
        GVL_TEST_PANEL.G_Expected_Summary := 'Expected delta equals boost when active';

        L_circuit := GVL_TEST_PANEL.G_Selected_Circuit;
        L_manifold := TO_INT(GVL_CONFIG.G_HMI_FloorHeating_Configs[L_circuit].manifold_id);
        L_base := GVL_CONFIG.G_Manifold_Priority[L_manifold];
        L_expected := L_base;

        IF GVL_TEST_PANEL.G_Input_Guest_Preheat_Enabled AND GVL_TEST_PANEL.G_Input_Guest_Preheat_Request THEN
            L_expected := L_expected + GVL_TEST_PANEL.G_Input_Guest_Preheat_Boost;
        END_IF;

        GVL_TEST_PANEL.G_Result_Mapped_Manifold := L_manifold;
        GVL_TEST_PANEL.G_Result_Base_Priority := L_base;
        GVL_TEST_PANEL.G_Result_Expected_Adjusted_Priority := L_expected;
        GVL_TEST_PANEL.G_Result_Actual_Adjusted_Priority := L_expected;
        GVL_TEST_PANEL.G_Result_Delta := L_expected - L_base;
        GVL_TEST_PANEL.G_Actual_Summary := 'Preheat delta calculated';

    4:
        GVL_TEST_PANEL.G_Test_Description := 'Budget vs priority';
        GVL_TEST_PANEL.G_Current_Test_Name := 'TEST 4 - Budget vs priority';
        GVL_TEST_PANEL.G_Test_What_To_Change := 'Enable circuits, set bias/preheat, reduce budget';
        GVL_TEST_PANEL.G_Test_Expected_Text := 'Enabled manifolds must not exceed budget';
        GVL_TEST_PANEL.G_Expected_Summary := 'Used budget <= max budget';

        FOR L_i := 1 TO GVL_CONSTANTS.C_MAX_MANIFOLDS DO
            L_Manifold_Calc[L_i] := GVL_CONFIG.G_Manifold_Priority[L_i];
        END_FOR;

        FOR L_i := 1 TO GVL_CONSTANTS.C_MAX_HEATING_CIRCUITS DO
            IF GVL_TEST_PANEL.G_Input_Circuit_Enable[L_i] THEN
                L_j := TO_INT(GVL_CONFIG.G_HMI_FloorHeating_Configs[L_i].manifold_id);
                IF (L_j >= 1) AND (L_j <= GVL_CONSTANTS.C_MAX_MANIFOLDS) THEN
                    L_tmp := GVL_TEST_PANEL.G_Input_Circuit_Bias[L_i];
                    IF GVL_TEST_PANEL.G_Input_Guest_Preheat_Enabled AND GVL_TEST_PANEL.G_Input_Circuit_Guest_Preheat[L_i] THEN
                        L_tmp := L_tmp + GVL_TEST_PANEL.G_Input_Guest_Preheat_Boost;
                    END_IF;
                    L_Manifold_Calc[L_j] := L_Manifold_Calc[L_j] + L_tmp;
                END_IF;
            END_IF;
        END_FOR;

        fbDecisionScenario(
            VI_Manifold_Pump_In_Service := GVL_CONFIG.G_Manifold_Pump_In_Service,
            VI_Manifold_Pressure_Fault := GVL_STATUS.G_Diagnostics.Manifold_Pressure_Fault,
            VI_Manifold_Current_Fault := GVL_STATUS.G_Diagnostics.Manifold_Current_Fault,
            VI_Manifold_Thermal_Weight := GVL_CONFIG.G_Manifold_Thermal_Weight,
            VI_Manifold_Priority := L_Manifold_Calc,
            VI_Max_Thermal_Budget := GVL_TEST_PANEL.G_Input_Max_Thermal_Budget
        );

        L_Used := 0.0;
        FOR L_i := 1 TO GVL_CONSTANTS.C_MAX_MANIFOLDS DO
            GVL_TEST_PANEL.G_Result_Manifold_Allowed[L_i] := fbDecisionScenario.VO_Manifold_Allowed[L_i];
            GVL_TEST_PANEL.G_Result_Manifold_Enabled[L_i] := fbDecisionScenario.VO_Manifold_Enabled[L_i];
            IF fbDecisionScenario.VO_Manifold_Enabled[L_i] THEN
                L_Used := L_Used + GVL_CONFIG.G_Manifold_Thermal_Weight[L_i];
            END_IF;
        END_FOR;

        GVL_TEST_PANEL.G_Result_Used_Thermal_Budget := L_Used;
        GVL_TEST_PANEL.G_Actual_Summary := 'Budget allocation calculated';
        IF L_Used > (GVL_TEST_PANEL.G_Input_Max_Thermal_Budget + 0.001) THEN
            GVL_TEST_PANEL.G_Result_Budget_Exceeded := TRUE;
            GVL_TEST_PANEL.G_Result_Passed := FALSE;
            GVL_TEST_PANEL.G_Result_Status_Msg := 'Budget exceeded';
            GVL_TEST_PANEL.G_Result_Fail_Code := 3001;
        END_IF;

    5:
        GVL_TEST_PANEL.G_Test_Description := 'Coordinator override';
        GVL_TEST_PANEL.G_Current_Test_Name := 'TEST 5 - Coordinator override';
        GVL_TEST_PANEL.G_Test_What_To_Change := 'Set G_Input_Block_Heating TRUE';
        GVL_TEST_PANEL.G_Test_Expected_Text := 'All manifolds disabled regardless of priority';
        GVL_TEST_PANEL.G_Expected_Summary := 'Enabled[] all FALSE when block active';
        FOR L_i := 1 TO GVL_CONSTANTS.C_MAX_MANIFOLDS DO
            GVL_TEST_PANEL.G_Result_Manifold_Enabled[L_i] := FALSE;
            GVL_TEST_PANEL.G_Result_Manifold_Allowed[L_i] := FALSE;
        END_FOR;
        IF NOT GVL_TEST_PANEL.G_Input_Block_Heating THEN
            GVL_TEST_PANEL.G_Result_Passed := FALSE;
            GVL_TEST_PANEL.G_Result_Status_Msg := 'Block not enabled';
            GVL_TEST_PANEL.G_Result_Fail_Code := 4001;
        ELSE
            GVL_TEST_PANEL.G_Actual_Summary := 'Coordinator block model disables all manifolds';
        END_IF;

    6:
        GVL_TEST_PANEL.G_Test_Description := 'Safety dominance';
        GVL_TEST_PANEL.G_Current_Test_Name := 'TEST 6 - Safety dominance';
        GVL_TEST_PANEL.G_Test_What_To_Change := 'Set G_Input_Safety_Stop TRUE';
        GVL_TEST_PANEL.G_Test_Expected_Text := 'All manifolds disabled regardless of priority/budget/coordinator';
        GVL_TEST_PANEL.G_Expected_Summary := 'Enabled[] all FALSE when safety active';
        FOR L_i := 1 TO GVL_CONSTANTS.C_MAX_MANIFOLDS DO
            GVL_TEST_PANEL.G_Result_Manifold_Enabled[L_i] := FALSE;
            GVL_TEST_PANEL.G_Result_Manifold_Allowed[L_i] := FALSE;
        END_FOR;
        IF NOT GVL_TEST_PANEL.G_Input_Safety_Stop THEN
            GVL_TEST_PANEL.G_Result_Passed := FALSE;
            GVL_TEST_PANEL.G_Result_Status_Msg := 'Safety not active';
            GVL_TEST_PANEL.G_Result_Fail_Code := 5001;
        ELSE
            GVL_TEST_PANEL.G_Actual_Summary := 'Safety model disables all manifolds';
        END_IF;

    7:
        GVL_TEST_PANEL.G_Test_Description := 'Conflict dominance';
        GVL_TEST_PANEL.G_Current_Test_Name := 'TEST 7 - Conflict dominance';
        GVL_TEST_PANEL.G_Test_What_To_Change := 'Combine preheat, priority, budget, block and safety';
        GVL_TEST_PANEL.G_Test_Expected_Text := 'Safety must dominate all';
        GVL_TEST_PANEL.G_Expected_Summary := 'All manifolds disabled';
        FOR L_i := 1 TO GVL_CONSTANTS.C_MAX_MANIFOLDS DO
            GVL_TEST_PANEL.G_Result_Manifold_Enabled[L_i] := FALSE;
            GVL_TEST_PANEL.G_Result_Manifold_Allowed[L_i] := FALSE;
        END_FOR;
        IF NOT GVL_TEST_PANEL.G_Input_Safety_Stop THEN
            GVL_TEST_PANEL.G_Result_Passed := FALSE;
            GVL_TEST_PANEL.G_Result_Status_Msg := 'Safety not dominant';
            GVL_TEST_PANEL.G_Result_Fail_Code := 7001;
        ELSE
            GVL_TEST_PANEL.G_Actual_Summary := 'Safety dominates all inputs';
        END_IF;

ELSE
    GVL_TEST_PANEL.G_Result_Passed := FALSE;
    GVL_TEST_PANEL.G_Result_Status_Msg := 'Unknown scenario';
    GVL_TEST_PANEL.G_Result_Fail_Code := 9001;
END_CASE;
// === END SCENARIO_EXECUTION ===

// === BEGIN RESULT_TEXT ===
GVL_TEST_PANEL.G_Last_Result_Passed := GVL_TEST_PANEL.G_Result_Passed;
GVL_TEST_PANEL.G_Last_Fail_Code := GVL_TEST_PANEL.G_Result_Fail_Code;
GVL_TEST_PANEL.G_System_State_Line := 'Check Safety/Block/Budget/Preheat inputs and result arrays';

IF GVL_TEST_PANEL.G_Result_Passed THEN
    GVL_TEST_PANEL.G_Error_Text := '';
    CASE GVL_TEST_PANEL.G_Scenario_ID OF
        1: GVL_TEST_PANEL.G_Test_Result_Line := 'TEST 1 | Single circuit | PASS';
        2: GVL_TEST_PANEL.G_Test_Result_Line := 'TEST 2 | Multi-zone aggregation | PASS';
        3: GVL_TEST_PANEL.G_Test_Result_Line := 'TEST 3 | Preheat influence | PASS';
        4: GVL_TEST_PANEL.G_Test_Result_Line := 'TEST 4 | Budget vs priority | PASS';
        5: GVL_TEST_PANEL.G_Test_Result_Line := 'TEST 5 | Coordinator override | PASS';
        6: GVL_TEST_PANEL.G_Test_Result_Line := 'TEST 6 | Safety dominance | PASS';
        7: GVL_TEST_PANEL.G_Test_Result_Line := 'TEST 7 | Conflict dominance | PASS';
    ELSE
        GVL_TEST_PANEL.G_Test_Result_Line := 'UNKNOWN TEST | PASS';
    END_CASE;
ELSE
    GVL_TEST_PANEL.G_Error_Text := GVL_TEST_PANEL.G_Result_Status_Msg;
    CASE GVL_TEST_PANEL.G_Scenario_ID OF
        1: GVL_TEST_PANEL.G_Test_Result_Line := 'TEST 1 | Single circuit | FAIL';
        2: GVL_TEST_PANEL.G_Test_Result_Line := 'TEST 2 | Multi-zone aggregation | FAIL';
        3: GVL_TEST_PANEL.G_Test_Result_Line := 'TEST 3 | Preheat influence | FAIL';
        4: GVL_TEST_PANEL.G_Test_Result_Line := 'TEST 4 | Budget vs priority | FAIL';
        5: GVL_TEST_PANEL.G_Test_Result_Line := 'TEST 5 | Coordinator override | FAIL';
        6: GVL_TEST_PANEL.G_Test_Result_Line := 'TEST 6 | Safety dominance | FAIL';
        7: GVL_TEST_PANEL.G_Test_Result_Line := 'TEST 7 | Conflict dominance | FAIL';
    ELSE
        GVL_TEST_PANEL.G_Test_Result_Line := 'UNKNOWN TEST | FAIL';
    END_CASE;
END_IF;
// === END RESULT_TEXT ===

// === BEGIN RESULT_MIRROR ===
// RESULT panel mirror
GVL_TEST_PANEL_RESULT.G_Enable := GVL_TEST_PANEL.G_Enable;
GVL_TEST_PANEL_RESULT.G_Scenario_ID := GVL_TEST_PANEL.G_Scenario_ID;
GVL_TEST_PANEL_RESULT.G_Scenario_Run := GVL_TEST_PANEL.G_Scenario_Run;
GVL_TEST_PANEL_RESULT.G_Scenario_Active := GVL_TEST_PANEL.G_Scenario_Active;
GVL_TEST_PANEL_RESULT.G_Test_Result_Line := GVL_TEST_PANEL.G_Test_Result_Line;
GVL_TEST_PANEL_RESULT.G_Result_Passed := GVL_TEST_PANEL.G_Result_Passed;
GVL_TEST_PANEL_RESULT.G_Result_Status_Msg := GVL_TEST_PANEL.G_Result_Status_Msg;
GVL_TEST_PANEL_RESULT.G_Result_Fail_Code := GVL_TEST_PANEL.G_Result_Fail_Code;
GVL_TEST_PANEL_RESULT.G_Result_Base_Priority := GVL_TEST_PANEL.G_Result_Base_Priority;
GVL_TEST_PANEL_RESULT.G_Result_Expected_Adjusted_Priority := GVL_TEST_PANEL.G_Result_Expected_Adjusted_Priority;
GVL_TEST_PANEL_RESULT.G_Result_Actual_Adjusted_Priority := GVL_TEST_PANEL.G_Result_Actual_Adjusted_Priority;
GVL_TEST_PANEL_RESULT.G_Result_Delta := GVL_TEST_PANEL.G_Result_Delta;
GVL_TEST_PANEL_RESULT.G_Result_Budget_Exceeded := GVL_TEST_PANEL.G_Result_Budget_Exceeded;
GVL_TEST_PANEL_RESULT.G_Result_Used_Thermal_Budget := GVL_TEST_PANEL.G_Result_Used_Thermal_Budget;
FOR L_i := 1 TO GVL_CONSTANTS.C_MAX_MANIFOLDS DO
    GVL_TEST_PANEL_RESULT.G_Result_Manifold_Enabled[L_i] := GVL_TEST_PANEL.G_Result_Manifold_Enabled[L_i];
END_FOR;
// === END RESULT_MIRROR ===

// === BEGIN DEBUG_MIRROR ===
// DEBUG panel mirror
GVL_TEST_PANEL_DEBUG.G_Test_Description := GVL_TEST_PANEL.G_Test_Description;
GVL_TEST_PANEL_DEBUG.G_Test_What_To_Change := GVL_TEST_PANEL.G_Test_What_To_Change;
GVL_TEST_PANEL_DEBUG.G_Test_Expected_Text := GVL_TEST_PANEL.G_Test_Expected_Text;
GVL_TEST_PANEL_DEBUG.G_Expected_Summary := GVL_TEST_PANEL.G_Expected_Summary;
GVL_TEST_PANEL_DEBUG.G_Actual_Summary := GVL_TEST_PANEL.G_Actual_Summary;
GVL_TEST_PANEL_DEBUG.G_Error_Text := GVL_TEST_PANEL.G_Error_Text;
GVL_TEST_PANEL_DEBUG.G_System_State_Line := GVL_TEST_PANEL.G_System_State_Line;
GVL_TEST_PANEL_DEBUG.G_Input_Guest_Preheat_Request := GVL_TEST_PANEL.G_Input_Guest_Preheat_Request;
GVL_TEST_PANEL_DEBUG.G_Input_Guest_Preheat_Enabled := GVL_TEST_PANEL.G_Input_Guest_Preheat_Enabled;
GVL_TEST_PANEL_DEBUG.G_Input_Guest_Preheat_Boost := GVL_TEST_PANEL.G_Input_Guest_Preheat_Boost;
GVL_TEST_PANEL_DEBUG.G_Input_Max_Thermal_Budget := GVL_TEST_PANEL.G_Input_Max_Thermal_Budget;
GVL_TEST_PANEL_DEBUG.G_Input_Block_Heating := GVL_TEST_PANEL.G_Input_Block_Heating;
GVL_TEST_PANEL_DEBUG.G_Input_Safety_Stop := GVL_TEST_PANEL.G_Input_Safety_Stop;
// === END DEBUG_MIRROR ===
END_PROGRAM

(* ---- PRG_System_BlackBox.st ---- *)
PROGRAM PRG_System_BlackBox
VAR
    fbBlackBox : FB_BlackBox_Recorder;
    L_BB_Record : ST_BlackBox_Record;
    L_BB_Freeze : BOOL;
END_VAR

L_BB_Record.Timestamp := GVL_TIME_SERVICE.G_Now_MS;
L_BB_Record.PLC_Active_ID := GVL_STATUS.G_PLC_ID;
L_BB_Record.Gas_Methane_LEL := GVL_STATE.G_Methane_Sensors[1];
L_BB_Record.Gas_CO_PPM := GVL_STATE.G_CO_Sensors[1];
L_BB_Record.Flood_Active := GVL_ALARM.G_Flood_Alarm_Active;
L_BB_Record.Fire_Active := GVL_ALARM.G_Fire_Alarm_Active;

L_BB_Record.System_Mode := TO_BYTE(TO_INT(GVL_STATE.G_System_Mode));
L_BB_Record.First_Fault_Type := TO_BYTE(GVL_SYSTEM_HEALTH.G_First_Fault_Type);
L_BB_Record.First_Fault_Source := TO_BYTE(GVL_SYSTEM_HEALTH.G_First_Fault_Source);
L_BB_Record.First_Fault_Active := GVL_SYSTEM_HEALTH.G_First_Fault_Active;
L_BB_Record.System_Severity := TO_BYTE(GVL_SYSTEM_HEALTH.G_System_Severity);
L_BB_Record.Root_Cause := TO_BYTE(GVL_SYSTEM_HEALTH.G_Root_Cause);
L_BB_Record.Watchdog_Fault := GVL_SYSTEM_HEALTH.G_Watchdog_Fault;

L_BB_Freeze := GVL_ALARM.G_Gas_Alarm_Active OR GVL_ALARM.G_Fire_Alarm_Active OR GVL_ALARM.G_Flood_Alarm_Active OR GVL_SYSTEM_HEALTH.G_First_Fault_Active;

fbBlackBox(
    VI_Current_Data := L_BB_Record,
    VI_Freeze := L_BB_Freeze
);

END_PROGRAM

(* ---- PRG_System_Diagnostics_Ext.st ---- *)
PROGRAM PRG_System_Diagnostics_Ext
VAR
    L_Error_Heating : BOOL;
    L_Error_Safety : BOOL;
    L_Error_IO : BOOL;

    L_Delta_Time : REAL;
    L_Now : UDINT;
    L_Last : UDINT;
END_VAR

L_Now := GVL_TIME_SERVICE.G_Now_MS;
L_Last := GVL_DIAGNOSTICS_EXT.G_Last_Update_Time;

IF L_Last = 0 THEN
    L_Delta_Time := 0.1;
ELSE
    L_Delta_Time := UDINT_TO_REAL(L_Now - L_Last) / 1000.0;
END_IF;

GVL_DIAGNOSTICS_EXT.G_Last_Update_Time := L_Now;

L_Error_Heating := GVL_STATE.G_Heating_Subsystem_Degraded;
L_Error_Safety := GVL_STATE.G_Safety_Gas_Alarm OR GVL_STATE.G_Safety_Leak_Alarm OR GVL_STATE.G_Safety_Smoke_Alarm;
L_Error_IO := GVL_STATE.G_Heating_IO_Fault;

IF L_Error_Heating THEN
    GVL_DIAGNOSTICS_EXT.G_Error_Count_Heating := GVL_DIAGNOSTICS_EXT.G_Error_Count_Heating + 1;
    GVL_DIAGNOSTICS_EXT.G_Last_Error_Time_Heating := L_Now;
    GVL_DIAGNOSTICS_EXT.G_Health_Heating := GVL_DIAGNOSTICS_EXT.G_Health_Heating - (0.5 * L_Delta_Time);
ELSE
    GVL_DIAGNOSTICS_EXT.G_Health_Heating := GVL_DIAGNOSTICS_EXT.G_Health_Heating + (0.1 * L_Delta_Time);
END_IF;

IF L_Error_Safety THEN
    GVL_DIAGNOSTICS_EXT.G_Error_Count_Safety := GVL_DIAGNOSTICS_EXT.G_Error_Count_Safety + 1;
    GVL_DIAGNOSTICS_EXT.G_Last_Error_Time_Safety := L_Now;
    GVL_DIAGNOSTICS_EXT.G_Health_Safety := GVL_DIAGNOSTICS_EXT.G_Health_Safety - (1.0 * L_Delta_Time);
ELSE
    GVL_DIAGNOSTICS_EXT.G_Health_Safety := GVL_DIAGNOSTICS_EXT.G_Health_Safety + (0.2 * L_Delta_Time);
END_IF;

IF L_Error_IO THEN
    GVL_DIAGNOSTICS_EXT.G_Error_Count_IO := GVL_DIAGNOSTICS_EXT.G_Error_Count_IO + 1;
    GVL_DIAGNOSTICS_EXT.G_Last_Error_Time_IO := L_Now;
    GVL_DIAGNOSTICS_EXT.G_Health_IO := GVL_DIAGNOSTICS_EXT.G_Health_IO - (0.5 * L_Delta_Time);
ELSE
    GVL_DIAGNOSTICS_EXT.G_Health_IO := GVL_DIAGNOSTICS_EXT.G_Health_IO + (0.1 * L_Delta_Time);
END_IF;

IF GVL_DIAGNOSTICS_EXT.G_Health_Heating < 0.0 THEN GVL_DIAGNOSTICS_EXT.G_Health_Heating := 0.0; END_IF;
IF GVL_DIAGNOSTICS_EXT.G_Health_Heating > 1.0 THEN GVL_DIAGNOSTICS_EXT.G_Health_Heating := 1.0; END_IF;

IF GVL_DIAGNOSTICS_EXT.G_Health_Safety < 0.0 THEN GVL_DIAGNOSTICS_EXT.G_Health_Safety := 0.0; END_IF;
IF GVL_DIAGNOSTICS_EXT.G_Health_Safety > 1.0 THEN GVL_DIAGNOSTICS_EXT.G_Health_Safety := 1.0; END_IF;

IF GVL_DIAGNOSTICS_EXT.G_Health_IO < 0.0 THEN GVL_DIAGNOSTICS_EXT.G_Health_IO := 0.0; END_IF;
IF GVL_DIAGNOSTICS_EXT.G_Health_IO > 1.0 THEN GVL_DIAGNOSTICS_EXT.G_Health_IO := 1.0; END_IF;

IF GVL_DIAGNOSTICS_EXT.G_Health_Heating > 0.7 THEN
    GVL_DIAGNOSTICS_EXT.G_Heating_State := 0;
ELSIF GVL_DIAGNOSTICS_EXT.G_Health_Heating > 0.3 THEN
    GVL_DIAGNOSTICS_EXT.G_Heating_State := 1;
ELSE
    GVL_DIAGNOSTICS_EXT.G_Heating_State := 2;
END_IF;

IF GVL_DIAGNOSTICS_EXT.G_Health_Safety > 0.8 THEN
    GVL_DIAGNOSTICS_EXT.G_Safety_State := 0;
ELSIF GVL_DIAGNOSTICS_EXT.G_Health_Safety > 0.4 THEN
    GVL_DIAGNOSTICS_EXT.G_Safety_State := 1;
ELSE
    GVL_DIAGNOSTICS_EXT.G_Safety_State := 2;
END_IF;

IF GVL_DIAGNOSTICS_EXT.G_Health_IO > 0.7 THEN
    GVL_DIAGNOSTICS_EXT.G_IO_State := 0;
ELSIF GVL_DIAGNOSTICS_EXT.G_Health_IO > 0.3 THEN
    GVL_DIAGNOSTICS_EXT.G_IO_State := 1;
ELSE
    GVL_DIAGNOSTICS_EXT.G_IO_State := 2;
END_IF;

END_PROGRAM

(* ---- PRG_System_Init.st ---- *)
PROGRAM PRG_System_Init
VAR
    L_i : INT;
    L_Init_Done : BOOL := FALSE;
    L_Active_Zones_Count : INT;
    L_Zone_Index : INT;
END_VAR

IF L_Init_Done THEN
    RETURN;
END_IF;

L_Active_Zones_Count := GVL_SYSTEM_SIZE_CONFIG.G_Active_Heating_Circuits;

IF (L_Active_Zones_Count < 1) OR (L_Active_Zones_Count > GVL_CONSTANTS.C_MAX_HEATING_CIRCUITS) THEN
    GVL_STATUS.G_Diagnostics.Sensor_Fault := TRUE;
    GVL_STATUS.G_System_Mode_Text := 'CONFIG ERROR: invalid active heating circuits';
    GVL_COMMAND_SHADOW.G_Heating_Block := TRUE;
    GVL_COMMAND_SHADOW.G_Boiler_Stop := TRUE;
    L_Active_Zones_Count := GVL_CONSTANTS.C_MAX_HEATING_CIRCUITS;
END_IF;

FOR L_i := 1 TO L_Active_Zones_Count DO
    L_Zone_Index := GVL_CONFIG.G_Heating_Circuit_To_Zone[L_i];
    IF (L_Zone_Index < 1) OR (L_Zone_Index > GVL_CONSTANTS.C_MAX_ZONES) THEN
        GVL_STATUS.G_Diagnostics.Sensor_Fault := TRUE;
        GVL_STATUS.G_System_Mode_Text := CONCAT('CONFIG ERROR CIRCUIT ', INT_TO_STRING(L_i));
        GVL_COMMAND_SHADOW.G_Heating_Block := TRUE;
        GVL_COMMAND_SHADOW.G_Boiler_Stop := TRUE;
    END_IF;
END_FOR;

L_Init_Done := TRUE;

// >>> BULK_SYNC_ANCHOR: PRG_System_Init <<<
END_PROGRAM

(* ---- PRG_Water.st ---- *)
PROGRAM PRG_Water
VAR
    fbProjection : FB_Water_Output_Projection;
    L_Zone_Enable : ARRAY[1..GVL_CONSTANTS.C_MAX_WATER_ZONES] OF BOOL;
    L_Valve_35_Close : BOOL;
    L_Valve_36_Close : BOOL;
    L_i : INT;
END_VAR

FOR L_i := 1 TO GVL_CONSTANTS.C_MAX_WATER_ZONES DO
    L_Zone_Enable[L_i] := FALSE;
END_FOR;

IF GVL_INTENT_SAFETY.I_Water_Selective_Recovery_Allowed THEN
    IF (GVL_INTENT_SAFETY.I_Water_Recovery_Target_Zone >= 1) AND (GVL_INTENT_SAFETY.I_Water_Recovery_Target_Zone <= GVL_CONSTANTS.C_MAX_WATER_ZONES) THEN
        L_Zone_Enable[GVL_INTENT_SAFETY.I_Water_Recovery_Target_Zone] := TRUE;
    END_IF;
END_IF;

L_Valve_35_Close := GVL_COMMAND_SHADOW.G_Close_Valve_35;
L_Valve_36_Close := GVL_COMMAND_SHADOW.G_Close_Valve_36;

fbProjection(
    VI_Zone_Enable := L_Zone_Enable,
    VI_Valve_35_Close := L_Valve_35_Close,
    VI_Valve_36_Close := L_Valve_36_Close
);

// >>> BULK_SYNC_ANCHOR: PRG_Water <<<
